LIN {X 0,Y 401.58,Z 643.451,A -85,B 0,C 180,E1 -18913.491,E2 -18913.491} C_VEL
LIN {X 0,Y 402.309,Z 631.628,A -85,B 0,C 180,E1 -18914.623,E2 -18914.623} C_VEL
LIN {X 0,Y 403.111,Z 618.78,A -85,B 0,C 180,E1 -18915.625,E2 -18915.625} C_VEL
LIN {X 0,Y 403.802,Z 604.625,A -85,B 0,C 180,E1 -18916.502,E2 -18916.502} C_VEL
LIN {X 0,Y 404.446,Z 589.348,A -85,B 0,C 180,E1 -18917.22,E2 -18917.22} C_VEL
LIN {X 0,Y 404.999,Z 573.982,A -85,B 0,C 180,E1 -18917.715,E2 -18917.715} C_VEL
LIN {X 0,Y 407.837,Z 472.83,A -85,B 0,C 180,E1 -18920.256,E2 -18920.256} C_VEL
LIN {X 0,Y 405.076,Z 441.864,A -85,B 0,C 180,E1 -18921.136,E2 -18921.136} C_VEL
LIN {X 0,Y 404.994,Z 439.403,A -85,B 0,C 180,E1 -18921.232,E2 -18921.232} C_VEL
LIN {X 0,Y 406.943,Z 410.051,A -85,B 0,C 180,E1 -18925.079,E2 -18925.079} C_VEL
LIN {X 0,Y 408.958,Z 382.784,A -85,B 0,C 180,E1 -18928.658,E2 -18928.658} C_VEL
LIN {X 0,Y 405.49,Z 366.591,A -85,B 0,C 180,E1 -18930.997,E2 -18930.997} C_VEL
LIN {X 0,Y 401.287,Z 348.058,A -85,B 0,C 180,E1 -18933.747,E2 -18933.747} C_VEL
LIN {X 0,Y 401.239,Z 348.061,A -85,B 0,C 180,E1 -18936.58,E2 -18936.58} C_VEL
LIN {X 0,Y 401.222,Z 348.061,A -85,B 0,C 180,E1 -18939.813,E2 -18939.813} C_VEL
LIN {X 0,Y 401.236,Z 348.064,A -85,B 0,C 180,E1 -18942.909,E2 -18942.909} C_VEL
LIN {X 0,Y 401.28,Z 348.053,A -85,B 0,C 180,E1 -18945.716,E2 -18945.716} C_VEL
LIN {X 0,Y 401.214,Z 348.067,A -85,B 0,C 180,E1 -18948.652,E2 -18948.652} C_VEL
LIN {X 0,Y 401.253,Z 348.057,A -85,B 0,C 180,E1 -18951.771,E2 -18951.771} C_VEL
LIN {X 0,Y 401.255,Z 348.059,A -85,B 0,C 180,E1 -18955.13,E2 -18955.13} C_VEL
LIN {X 0,Y 401.243,Z 348.059,A -85,B 0,C 180,E1 -18958.803,E2 -18958.803} C_VEL
LIN {X 0,Y 401.259,Z 348.058,A -85,B 0,C 180,E1 -18961.88,E2 -18961.88} C_VEL
LIN {X 0,Y 401.254,Z 348.058,A -85,B 0,C 180,E1 -18965.232,E2 -18965.232} C_VEL
LIN {X 0,Y 401.256,Z 348.062,A -85,B 0,C 180,E1 -18968.495,E2 -18968.495} C_VEL
LIN {X 0,Y 401.293,Z 348.058,A -85,B 0,C 180,E1 -18971.689,E2 -18971.689} C_VEL
LIN {X 0,Y 401.284,Z 348.059,A -85,B 0,C 180,E1 -18972.24,E2 -18972.24} C_VEL
LIN {X 0,Y 404.072,Z 355.193,A -85,B 0,C 180,E1 -18972.535,E2 -18972.535} C_VEL
LIN {X 0,Y 412.124,Z 375.34,A -85,B 0,C 180,E1 -18973.336,E2 -18973.336} C_VEL
LIN {X 0,Y 410.823,Z 454.396,A -85,B 0,C 180,E1 -18974.708,E2 -18974.708} C_VEL
LIN {X 0,Y 410.699,Z 471.641,A -85,B 0,C 180,E1 -18975.083,E2 -18975.083} C_VEL
LIN {X 0,Y 410.292,Z 486.19,A -85,B 0,C 180,E1 -18975.605,E2 -18975.605} C_VEL
LIN {X 0,Y 409.658,Z 499.427,A -85,B 0,C 180,E1 -18976.276,E2 -18976.276} C_VEL
LIN {X 0,Y 408.783,Z 512.277,A -85,B 0,C 180,E1 -18977.129,E2 -18977.129} C_VEL
LIN {X 0,Y 407.855,Z 525.041,A -85,B 0,C 180,E1 -18978.214,E2 -18978.214} C_VEL
LIN {X 0,Y 406.772,Z 536.867,A -85,B 0,C 180,E1 -18979.458,E2 -18979.458} C_VEL
LIN {X 0,Y 405.528,Z 547.412,A -85,B 0,C 180,E1 -18980.807,E2 -18980.807} C_VEL
LIN {X 0,Y 404.408,Z 556.91,A -85,B 0,C 180,E1 -18982.286,E2 -18982.286} C_VEL
LIN {X 0,Y 403.349,Z 564.807,A -85,B 0,C 180,E1 -18983.769,E2 -18983.769} C_VEL
LIN {X 0,Y 402.397,Z 572.372,A -85,B 0,C 180,E1 -18985.508,E2 -18985.508} C_VEL
LIN {X 0,Y 401.791,Z 577.649,A -85,B 0,C 180,E1 -18987.002,E2 -18987.002} C_VEL
LIN {X 0,Y 401.183,Z 583.211,A -85,B 0,C 180,E1 -18989,E2 -18989} C_VEL
LIN {X 0,Y 400.805,Z 587.257,A -85,B 0,C 180,E1 -18991.002,E2 -18991.002} C_VEL
LIN {X 0,Y 400.584,Z 589.922,A -85,B 0,C 180,E1 -18993.007,E2 -18993.007} C_VEL
LIN {X 0,Y 400.657,Z 591.257,A -85,B 0,C 180,E1 -18995.015,E2 -18995.015} C_VEL
LIN {X 0,Y 400.827,Z 591.305,A -85,B 0,C 180,E1 -18997.026,E2 -18997.026} C_VEL
LIN {X 0,Y 401.166,Z 590.052,A -85,B 0,C 180,E1 -18999.041,E2 -18999.041} C_VEL
LIN {X 0,Y 401.726,Z 587.461,A -85,B 0,C 180,E1 -19001.058,E2 -19001.058} C_VEL
LIN {X 0,Y 402.683,Z 583.437,A -85,B 0,C 180,E1 -19003.069,E2 -19003.069} C_VEL
LIN {X 0,Y 403.855,Z 577.868,A -85,B 0,C 180,E1 -19005.08,E2 -19005.08} C_VEL
LIN {X 0,Y 404.901,Z 572.55,A -85,B 0,C 180,E1 -19006.585,E2 -19006.585} C_VEL
LIN {X 0,Y 406.377,Z 564.566,A -85,B 0,C 180,E1 -19008.407,E2 -19008.407} C_VEL
LIN {X 0,Y 408.022,Z 555.415,A -85,B 0,C 180,E1 -19010.081,E2 -19010.081} C_VEL
LIN {X 0,Y 409.614,Z 545.412,A -85,B 0,C 180,E1 -19011.571,E2 -19011.571} C_VEL
LIN {X 0,Y 411.2,Z 534.021,A -85,B 0,C 180,E1 -19012.948,E2 -19012.948} C_VEL
LIN {X 0,Y 412.585,Z 522.901,A -85,B 0,C 180,E1 -19014.045,E2 -19014.045} C_VEL
LIN {X 0,Y 413.931,Z 510.55,A -85,B 0,C 180,E1 -19015.027,E2 -19015.027} C_VEL
LIN {X 0,Y 414.787,Z 497.822,A -85,B 0,C 180,E1 -19015.842,E2 -19015.842} C_VEL
LIN {X 0,Y 415.567,Z 483.487,A -85,B 0,C 180,E1 -19016.527,E2 -19016.527} C_VEL
LIN {X 0,Y 415.988,Z 469.059,A -85,B 0,C 180,E1 -19017.004,E2 -19017.004} C_VEL
LIN {X 0,Y 416.665,Z 431.837,A -85,B 0,C 180,E1 -19017.69,E2 -19017.69} C_VEL
LIN {X 0,Y 416.122,Z 426.037,A -85,B 0,C 180,E1 -19017.834,E2 -19017.834} C_VEL
LIN {X 0,Y 411.482,Z 407.365,A -85,B 0,C 180,E1 -19018.5,E2 -19018.5} C_VEL
LIN {X 0,Y 411.102,Z 401.561,A -85,B 0,C 180,E1 -19018.638,E2 -19018.638} C_VEL
LIN {X 0,Y 411.271,Z 385.01,A -85,B 0,C 180,E1 -19018.943,E2 -19018.943} C_VEL
LIN {X 0,Y 402.695,Z 366.36,A -85,B 0,C 180,E1 -19019.927,E2 -19019.927} C_VEL
LIN {X 0,Y 394.318,Z 349.692,A -85,B 0,C 180,E1 -19020.909,E2 -19020.909} C_VEL
LIN {X 0,Y 394.183,Z 348.941,A -85,B 0,C 180,E1 -19020.969,E2 -19020.969} C_VEL
LIN {X 0,Y 394.127,Z 348.949,A -85,B 0,C 180,E1 -19024.66,E2 -19024.66} C_VEL
LIN {X 0,Y 394.153,Z 348.945,A -85,B 0,C 180,E1 -19027.172,E2 -19027.172} C_VEL
LIN {X 0,Y 394.132,Z 348.949,A -85,B 0,C 180,E1 -19030.165,E2 -19030.165} C_VEL
LIN {X 0,Y 394.138,Z 348.951,A -85,B 0,C 180,E1 -19033.876,E2 -19033.876} C_VEL
LIN {X 0,Y 394.145,Z 348.946,A -85,B 0,C 180,E1 -19036.771,E2 -19036.771} C_VEL
LIN {X 0,Y 394.134,Z 348.944,A -85,B 0,C 180,E1 -19040.224,E2 -19040.224} C_VEL
LIN {X 0,Y 394.148,Z 348.906,A -85,B 0,C 180,E1 -19043.102,E2 -19043.102} C_VEL
LIN {X 0,Y 394.15,Z 348.941,A -85,B 0,C 180,E1 -19046.641,E2 -19046.641} C_VEL
LIN {X 0,Y 394.173,Z 348.935,A -85,B 0,C 180,E1 -19050.161,E2 -19050.161} C_VEL
LIN {X 0,Y 394.207,Z 348.929,A -85,B 0,C 180,E1 -19053.627,E2 -19053.627} C_VEL
LIN {X 0,Y 394.168,Z 348.942,A -85,B 0,C 180,E1 -19056.986,E2 -19056.986} C_VEL
LIN {X 0,Y 394.202,Z 348.929,A -85,B 0,C 180,E1 -19058.535,E2 -19058.535} C_VEL
LIN {X 0,Y 400.317,Z 371.331,A -85,B 0,C 180,E1 -19059.301,E2 -19059.301} C_VEL
LIN {X 0,Y 398.077,Z 464.711,A -85,B 0,C 180,E1 -19061.671,E2 -19061.671} C_VEL
LIN {X 0,Y 397.816,Z 479.463,A -85,B 0,C 180,E1 -19062.218,E2 -19062.218} C_VEL
LIN {X 0,Y 397.322,Z 493.984,A -85,B 0,C 180,E1 -19062.957,E2 -19062.957} C_VEL
LIN {X 0,Y 396.777,Z 507.71,A -85,B 0,C 180,E1 -19063.856,E2 -19063.856} C_VEL
LIN {X 0,Y 396.137,Z 520.276,A -85,B 0,C 180,E1 -19064.882,E2 -19064.882} C_VEL
LIN {X 0,Y 395.506,Z 533.102,A -85,B 0,C 180,E1 -19066.167,E2 -19066.167} C_VEL
LIN {X 0,Y 395.015,Z 544.496,A -85,B 0,C 180,E1 -19067.548,E2 -19067.548} C_VEL
LIN {X 0,Y 394.447,Z 554.452,A -85,B 0,C 180,E1 -19068.995,E2 -19068.995} C_VEL
LIN {X 0,Y 393.925,Z 563.283,A -85,B 0,C 180,E1 -19070.533,E2 -19070.533} C_VEL
LIN {X 0,Y 393.535,Z 571.747,A -85,B 0,C 180,E1 -19072.328,E2 -19072.328} C_VEL
LIN {X 0,Y 393.339,Z 577.712,A -85,B 0,C 180,E1 -19073.866,E2 -19073.866} C_VEL
LIN {X 0,Y 393.339,Z 584.025,A -85,B 0,C 180,E1 -19075.915,E2 -19075.915} C_VEL
LIN {X 0,Y 393.351,Z 587.625,A -85,B 0,C 180,E1 -19077.448,E2 -19077.448} C_VEL
LIN {X 0,Y 393.465,Z 590.375,A -85,B 0,C 180,E1 -19078.98,E2 -19078.98} C_VEL
LIN {X 0,Y 393.85,Z 592.716,A -85,B 0,C 180,E1 -19081.019,E2 -19081.019} C_VEL
LIN {X 0,Y 394.504,Z 593.628,A -85,B 0,C 180,E1 -19083.053,E2 -19083.053} C_VEL
LIN {X 0,Y 395.419,Z 593.116,A -85,B 0,C 180,E1 -19085.081,E2 -19085.081} C_VEL
LIN {X 0,Y 396.591,Z 591.142,A -85,B 0,C 180,E1 -19087.101,E2 -19087.101} C_VEL
LIN {X 0,Y 397.274,Z 589.601,A -85,B 0,C 180,E1 -19088.108,E2 -19088.108} C_VEL
LIN {X 0,Y 399.178,Z 585.289,A -85,B 0,C 180,E1 -19090.106,E2 -19090.106} C_VEL
LIN {X 0,Y 400.768,Z 580.992,A -85,B 0,C 180,E1 -19091.595,E2 -19091.595} C_VEL
LIN {X 0,Y 402.678,Z 574.711,A -85,B 0,C 180,E1 -19093.325,E2 -19093.325} C_VEL
LIN {X 0,Y 404.905,Z 566.861,A -85,B 0,C 180,E1 -19095.039,E2 -19095.039} C_VEL
LIN {X 0,Y 406.955,Z 558.64,A -85,B 0,C 180,E1 -19096.499,E2 -19096.499} C_VEL
LIN {X 0,Y 409.19,Z 548.719,A -85,B 0,C 180,E1 -19097.946,E2 -19097.946} C_VEL
LIN {X 0,Y 411.656,Z 536.579,A -85,B 0,C 180,E1 -19099.378,E2 -19099.378} C_VEL
LIN {X 0,Y 413.904,Z 524.167,A -85,B 0,C 180,E1 -19100.557,E2 -19100.557} C_VEL
LIN {X 0,Y 415.905,Z 509.912,A -85,B 0,C 180,E1 -19101.651,E2 -19101.651} C_VEL
LIN {X 0,Y 417.437,Z 495.791,A -85,B 0,C 180,E1 -19102.508,E2 -19102.508} C_VEL
LIN {X 0,Y 418.537,Z 482.493,A -85,B 0,C 180,E1 -19103.123,E2 -19103.123} C_VEL
LIN {X 0,Y 419.857,Z 461.411,A -85,B 0,C 180,E1 -19103.831,E2 -19103.831} C_VEL
LIN {X 0,Y 425.647,Z 397.413,A -85,B 0,C 180,E1 -19105.699,E2 -19105.699} C_VEL
LIN {X 0,Y 420.947,Z 388.333,A -85,B 0,C 180,E1 -19106.87,E2 -19106.87} C_VEL
LIN {X 0,Y 415.066,Z 378.237,A -85,B 0,C 180,E1 -19108.46,E2 -19108.46} C_VEL
LIN {X 0,Y 411.495,Z 373.014,A -85,B 0,C 180,E1 -19109.492,E2 -19109.492} C_VEL
LIN {X 0,Y 408.951,Z 369.218,A -85,B 0,C 180,E1 -19110.302,E2 -19110.302} C_VEL
LIN {X 0,Y 406.363,Z 365.403,A -85,B 0,C 180,E1 -19111.188,E2 -19111.188} C_VEL
LIN {X 0,Y 403.453,Z 361.802,A -85,B 0,C 180,E1 -19112.251,E2 -19112.251} C_VEL
LIN {X 0,Y 402.379,Z 359.935,A -85,B 0,C 180,E1 -19112.701,E2 -19112.701} C_VEL
LIN {X 0,Y 399.857,Z 357.401,A -85,B 0,C 180,E1 -19113.756,E2 -19113.756} C_VEL
LIN {X 0,Y 398.478,Z 354.589,A -85,B 0,C 180,E1 -19114.493,E2 -19114.493} C_VEL
LIN {X 0,Y 395.991,Z 352.852,A -85,B 0,C 180,E1 -19115.712,E2 -19115.712} C_VEL
LIN {X 0,Y 394.311,Z 349.707,A -85,B 0,C 180,E1 -19117.154,E2 -19117.154} C_VEL
LIN {X 0,Y 394.188,Z 348.932,A -85,B 0,C 180,E1 -19117.488,E2 -19117.488} C_VEL
LIN {X 0,Y 394.141,Z 348.938,A -85,B 0,C 180,E1 -19121.113,E2 -19121.113} C_VEL
LIN {X 0,Y 394.174,Z 348.938,A -85,B 0,C 180,E1 -19124.7,E2 -19124.7} C_VEL
LIN {X 0,Y 394.149,Z 348.943,A -85,B 0,C 180,E1 -19128.278,E2 -19128.278} C_VEL
LIN {X 0,Y 394.165,Z 349.108,A -85,B 0,C 180,E1 -19129.409,E2 -19129.409} C_VEL
LIN {X 0,Y 395.196,Z 351.875,A -85,B 0,C 180,E1 -19130.436,E2 -19130.436} C_VEL
LIN {X 0,Y 397.598,Z 354.181,A -85,B 0,C 180,E1 -19131.854,E2 -19131.854} C_VEL
LIN {X 0,Y 398.536,Z 354.801,A -85,B 0,C 180,E1 -19132.321,E2 -19132.321} C_VEL
LIN {X 0,Y 399.934,Z 357.773,A -85,B 0,C 180,E1 -19133.146,E2 -19133.146} C_VEL
LIN {X 0,Y 400.838,Z 359.111,A -85,B 0,C 180,E1 -19133.603,E2 -19133.603} C_VEL
LIN {X 0,Y 405.1,Z 371.833,A -85,B 0,C 180,E1 -19135.918,E2 -19135.918} C_VEL
LIN {X 0,Y 409.584,Z 385.954,A -85,B 0,C 180,E1 -19137.895,E2 -19137.895} C_VEL
LIN {X 0,Y 410.898,Z 390.124,A -85,B 0,C 180,E1 -19138.422,E2 -19138.422} C_VEL
LIN {X 0,Y 412.58,Z 396.205,A -85,B 0,C 180,E1 -19139.099,E2 -19139.099} C_VEL
LIN {X 0,Y 414.9,Z 416.547,A -85,B 0,C 180,E1 -19140.564,E2 -19140.564} C_VEL
LIN {X 0,Y 417.082,Z 438.07,A -85,B 0,C 180,E1 -19141.924,E2 -19141.924} C_VEL
LIN {X 0,Y 418.558,Z 458.629,A -85,B 0,C 180,E1 -19143.047,E2 -19143.047} C_VEL
LIN {X 0,Y 419,Z 480.558,A -85,B 0,C 180,E1 -19144.021,E2 -19144.021} C_VEL
LIN {X 0,Y 416.342,Z 513.747,A -85,B 0,C 180,E1 -19144.995,E2 -19144.995} C_VEL
LIN {X 0,Y 413.523,Z 547.21,A -85,B 0,C 180,E1 -19145.98,E2 -19145.98} C_VEL
LIN {X 0,Y 411.488,Z 563.008,A -85,B 0,C 180,E1 -19146.62,E2 -19146.62} C_VEL
LIN {X 0,Y 408.946,Z 578.628,A -85,B 0,C 180,E1 -19147.465,E2 -19147.465} C_VEL
LIN {X 0,Y 406.192,Z 593.435,A -85,B 0,C 180,E1 -19148.504,E2 -19148.504} C_VEL
LIN {X 0,Y 403.496,Z 606.656,A -85,B 0,C 180,E1 -19149.684,E2 -19149.684} C_VEL
LIN {X 0,Y 400.718,Z 619.767,A -85,B 0,C 180,E1 -19151.133,E2 -19151.133} C_VEL
LIN {X 0,Y 398.386,Z 630.692,A -85,B 0,C 180,E1 -19152.609,E2 -19152.609} C_VEL
LIN {X 0,Y 396.45,Z 639.832,A -85,B 0,C 180,E1 -19154.106,E2 -19154.106} C_VEL
LIN {X 0,Y 394.809,Z 648.723,A -85,B 0,C 180,E1 -19155.88,E2 -19155.88} C_VEL
LIN {X 0,Y 393.743,Z 656.054,A -85,B 0,C 180,E1 -19157.674,E2 -19157.674} C_VEL
LIN {X 0,Y 393.485,Z 658.116,A -85,B 0,C 180,E1 -19158.171,E2 -19158.171} C_VEL
LIN {X 0,Y 392.987,Z 667.205,A -85,B 0,C 180,E1 -19159.473,E2 -19159.473} C_VEL
LIN {X 0,Y 392.568,Z 676.261,A -85,B 0,C 180,E1 -19161.018,E2 -19161.018} C_VEL
LIN {X 0,Y 392.231,Z 684.852,A -85,B 0,C 180,E1 -19162.819,E2 -19162.819} C_VEL
LIN {X 0,Y 392.082,Z 690.842,A -85,B 0,C 180,E1 -19164.361,E2 -19164.361} C_VEL
LIN {X 0,Y 391.975,Z 695.673,A -85,B 0,C 180,E1 -19165.901,E2 -19165.901} C_VEL
LIN {X 0,Y 391.913,Z 699.461,A -85,B 0,C 180,E1 -19167.439,E2 -19167.439} C_VEL
LIN {X 0,Y 391.91,Z 702.341,A -85,B 0,C 180,E1 -19168.976,E2 -19168.976} C_VEL
LIN {X 0,Y 391.919,Z 703.757,A -85,B 0,C 180,E1 -19170,E2 -19170} C_VEL
LIN {X 0,Y 391.891,Z 705.465,A -85,B 0,C 180,E1 -19172.048,E2 -19172.048} C_VEL
LIN {X 0,Y 391.96,Z 705.706,A -85,B 0,C 180,E1 -19174.099,E2 -19174.099} C_VEL
LIN {X 0,Y 392.331,Z 704.501,A -85,B 0,C 180,E1 -19176.149,E2 -19176.149} C_VEL
LIN {X 0,Y 393.018,Z 701.849,A -85,B 0,C 180,E1 -19178.197,E2 -19178.197} C_VEL
LIN {X 0,Y 393.984,Z 697.662,A -85,B 0,C 180,E1 -19180.241,E2 -19180.241} C_VEL
LIN {X 0,Y 395.723,Z 691.846,A -85,B 0,C 180,E1 -19182.263,E2 -19182.263} C_VEL
LIN {X 0,Y 397.333,Z 684.798,A -85,B 0,C 180,E1 -19184.17,E2 -19184.17} C_VEL
LIN {X 0,Y 399.284,Z 677.293,A -85,B 0,C 180,E1 -19185.778,E2 -19185.778} C_VEL
LIN {X 0,Y 401.742,Z 667.387,A -85,B 0,C 180,E1 -19187.503,E2 -19187.503} C_VEL
LIN {X 0,Y 404.089,Z 657.084,A -85,B 0,C 180,E1 -19188.966,E2 -19188.966} C_VEL
LIN {X 0,Y 406.809,Z 644.673,A -85,B 0,C 180,E1 -19190.406,E2 -19190.406} C_VEL
LIN {X 0,Y 409.335,Z 632.032,A -85,B 0,C 180,E1 -19191.586,E2 -19191.586} C_VEL
LIN {X 0,Y 411.507,Z 619.821,A -85,B 0,C 180,E1 -19192.518,E2 -19192.518} C_VEL
LIN {X 0,Y 413.893,Z 604.525,A -85,B 0,C 180,E1 -19193.434,E2 -19193.434} C_VEL
LIN {X 0,Y 415.936,Z 589.429,A -85,B 0,C 180,E1 -19194.103,E2 -19194.103} C_VEL
LIN {X 0,Y 418.104,Z 566.637,A -85,B 0,C 180,E1 -19194.816,E2 -19194.816} C_VEL
LIN {X 0,Y 425.848,Z 486.064,A -85,B 0,C 180,E1 -19197.224,E2 -19197.224} C_VEL
LIN {X 0,Y 426.185,Z 476.939,A -85,B 0,C 180,E1 -19197.591,E2 -19197.591} C_VEL
LIN {X 0,Y 425.687,Z 457.567,A -85,B 0,C 180,E1 -19198.602,E2 -19198.602} C_VEL
LIN {X 0,Y 424.826,Z 444.628,A -85,B 0,C 180,E1 -19199.408,E2 -19199.408} C_VEL
LIN {X 0,Y 424.35,Z 436.844,A -85,B 0,C 180,E1 -19199.955,E2 -19199.955} C_VEL
LIN {X 0,Y 426.009,Z 420.687,A -85,B 0,C 180,E1 -19201.593,E2 -19201.593} C_VEL
LIN {X 0,Y 427.546,Z 409.077,A -85,B 0,C 180,E1 -19202.914,E2 -19202.914} C_VEL
LIN {X 0,Y 427.531,Z 403.537,A -85,B 0,C 180,E1 -19203.851,E2 -19203.851} C_VEL
LIN {X 0,Y 426.297,Z 400.847,A -85,B 0,C 180,E1 -19204.76,E2 -19204.76} C_VEL
LIN {X 0,Y 424.019,Z 397.104,A -85,B 0,C 180,E1 -19206.491,E2 -19206.491} C_VEL
LIN {X 0,Y 422.633,Z 394.946,A -85,B 0,C 180,E1 -19207.822,E2 -19207.822} C_VEL
LIN {X 0,Y 420.894,Z 392.809,A -85,B 0,C 180,E1 -19210.046,E2 -19210.046} C_VEL
LIN {X 0,Y 420.043,Z 392.103,A -85,B 0,C 180,E1 -19211.838,E2 -19211.838} C_VEL
LIN {X 0,Y 419.719,Z 392.284,A -85,B 0,C 180,E1 -19214.143,E2 -19214.143} C_VEL
LIN {X 0,Y 419.855,Z 393.5,A -85,B 0,C 180,E1 -19215.838,E2 -19215.838} C_VEL
LIN {X 0,Y 420.591,Z 396.611,A -85,B 0,C 180,E1 -19218.229,E2 -19218.229} C_VEL
LIN {X 0,Y 421.525,Z 400.483,A -85,B 0,C 180,E1 -19220.238,E2 -19220.238} C_VEL
LIN {X 0,Y 422.633,Z 405.321,A -85,B 0,C 180,E1 -19222.178,E2 -19222.178} C_VEL
LIN {X 0,Y 423.731,Z 411.286,A -85,B 0,C 180,E1 -19224.095,E2 -19224.095} C_VEL
LIN {X 0,Y 424.745,Z 419.525,A -85,B 0,C 180,E1 -19226.25,E2 -19226.25} C_VEL
LIN {X 0,Y 424.873,Z 421.549,A -85,B 0,C 180,E1 -19226.716,E2 -19226.716} C_VEL
LIN {X 0,Y 420.776,Z 439.481,A -85,B 0,C 180,E1 -19229.434,E2 -19229.434} C_VEL
LIN {X 0,Y 423.204,Z 456.319,A -85,B 0,C 180,E1 -19230.818,E2 -19230.818} C_VEL
LIN {X 0,Y 425.126,Z 471.437,A -85,B 0,C 180,E1 -19231.888,E2 -19231.888} C_VEL
LIN {X 0,Y 426.272,Z 485.082,A -85,B 0,C 180,E1 -19232.701,E2 -19232.701} C_VEL
LIN {X 0,Y 418.787,Z 563.538,A -85,B 0,C 180,E1 -19235.019,E2 -19235.019} C_VEL
LIN {X 0,Y 416.753,Z 585.213,A -85,B 0,C 180,E1 -19235.684,E2 -19235.684} C_VEL
LIN {X 0,Y 414.717,Z 600.648,A -85,B 0,C 180,E1 -19236.351,E2 -19236.351} C_VEL
LIN {X 0,Y 412.612,Z 614.555,A -85,B 0,C 180,E1 -19237.15,E2 -19237.15} C_VEL
LIN {X 0,Y 410.394,Z 627.255,A -85,B 0,C 180,E1 -19238.078,E2 -19238.078} C_VEL
LIN {X 0,Y 407.829,Z 640.307,A -85,B 0,C 180,E1 -19239.254,E2 -19239.254} C_VEL
LIN {X 0,Y 405.259,Z 652.194,A -85,B 0,C 180,E1 -19240.567,E2 -19240.567} C_VEL
LIN {X 0,Y 402.728,Z 663,A -85,B 0,C 180,E1 -19242.018,E2 -19242.018} C_VEL
LIN {X 0,Y 400.549,Z 671.981,A -85,B 0,C 180,E1 -19243.491,E2 -19243.491} C_VEL
LIN {X 0,Y 398.442,Z 680.08,A -85,B 0,C 180,E1 -19245.089,E2 -19245.089} C_VEL
LIN {X 0,Y 396.813,Z 686.833,A -85,B 0,C 180,E1 -19246.734,E2 -19246.734} C_VEL
LIN {X 0,Y 395.371,Z 691.981,A -85,B 0,C 180,E1 -19248.245,E2 -19248.245} C_VEL
LIN {X 0,Y 393.93,Z 697.271,A -85,B 0,C 180,E1 -19250.275,E2 -19250.275} C_VEL
LIN {X 0,Y 393.122,Z 700.254,A -85,B 0,C 180,E1 -19251.805,E2 -19251.805} C_VEL
LIN {X 0,Y 392.364,Z 702.892,A -85,B 0,C 180,E1 -19253.851,E2 -19253.851} C_VEL
LIN {X 0,Y 391.948,Z 704.083,A -85,B 0,C 180,E1 -19255.901,E2 -19255.901} C_VEL
LIN {X 0,Y 391.803,Z 703.841,A -85,B 0,C 180,E1 -19257.951,E2 -19257.951} C_VEL
LIN {X 0,Y 391.821,Z 702.153,A -85,B 0,C 180,E1 -19260,E2 -19260} C_VEL
LIN {X 0,Y 391.848,Z 698.975,A -85,B 0,C 180,E1 -19262.049,E2 -19262.049} C_VEL
LIN {X 0,Y 391.881,Z 695.519,A -85,B 0,C 180,E1 -19263.587,E2 -19263.587} C_VEL
LIN {X 0,Y 391.993,Z 691.113,A -85,B 0,C 180,E1 -19265.126,E2 -19265.126} C_VEL
LIN {X 0,Y 392.192,Z 684.591,A -85,B 0,C 180,E1 -19266.924,E2 -19266.924} C_VEL
LIN {X 0,Y 392.518,Z 676.425,A -85,B 0,C 180,E1 -19268.725,E2 -19268.725} C_VEL
LIN {X 0,Y 392.94,Z 667.866,A -85,B 0,C 180,E1 -19270.269,E2 -19270.269} C_VEL
LIN {X 0,Y 393.625,Z 657.306,A -85,B 0,C 180,E1 -19271.844,E2 -19271.844} C_VEL
LIN {X 0,Y 394.334,Z 646.08,A -85,B 0,C 180,E1 -19273.221,E2 -19273.221} C_VEL
LIN {X 0,Y 395.082,Z 633.392,A -85,B 0,C 180,E1 -19274.503,E2 -19274.503} C_VEL
LIN {X 0,Y 395.913,Z 621.035,A -85,B 0,C 180,E1 -19275.521,E2 -19275.521} C_VEL
LIN {X 0,Y 396.666,Z 607.579,A -85,B 0,C 180,E1 -19276.412,E2 -19276.412} C_VEL
LIN {X 0,Y 397.25,Z 593.912,A -85,B 0,C 180,E1 -19277.112,E2 -19277.112} C_VEL
LIN {X 0,Y 397.813,Z 578.573,A -85,B 0,C 180,E1 -19277.683,E2 -19277.683} C_VEL
LIN {X 0,Y 400.841,Z 473.137,A -85,B 0,C 180,E1 -19280.423,E2 -19280.423} C_VEL
LIN {X 0,Y 398.096,Z 441.756,A -85,B 0,C 180,E1 -19281.333,E2 -19281.333} C_VEL
LIN {X 0,Y 398.002,Z 439.421,A -85,B 0,C 180,E1 -19281.426,E2 -19281.426} C_VEL
LIN {X 0,Y 399.917,Z 411.459,A -85,B 0,C 180,E1 -19285.134,E2 -19285.134} C_VEL
LIN {X 0,Y 401.909,Z 385.067,A -85,B 0,C 180,E1 -19288.638,E2 -19288.638} C_VEL
LIN {X 0,Y 401.665,Z 382.149,A -85,B 0,C 180,E1 -19289.048,E2 -19289.048} C_VEL
LIN {X 0,Y 396.805,Z 360.231,A -85,B 0,C 180,E1 -19292.274,E2 -19292.274} C_VEL
LIN {X 0,Y 394.258,Z 348.932,A -85,B 0,C 180,E1 -19293.988,E2 -19293.988} C_VEL
LIN {X 0,Y 394.184,Z 348.945,A -85,B 0,C 180,E1 -19297.169,E2 -19297.169} C_VEL
LIN {X 0,Y 394.169,Z 348.938,A -85,B 0,C 180,E1 -19300.171,E2 -19300.171} C_VEL
LIN {X 0,Y 394.222,Z 348.933,A -85,B 0,C 180,E1 -19303.864,E2 -19303.864} C_VEL
LIN {X 0,Y 394.181,Z 348.941,A -85,B 0,C 180,E1 -19306.766,E2 -19306.766} C_VEL
LIN {X 0,Y 394.175,Z 348.938,A -85,B 0,C 180,E1 -19310.229,E2 -19310.229} C_VEL
LIN {X 0,Y 394.187,Z 348.938,A -85,B 0,C 180,E1 -19313.095,E2 -19313.095} C_VEL
LIN {X 0,Y 394.2,Z 348.936,A -85,B 0,C 180,E1 -19315.347,E2 -19315.347} C_VEL
LIN {X 0,Y 394.192,Z 348.937,A -85,B 0,C 180,E1 -19318.982,E2 -19318.982} C_VEL
LIN {X 0,Y 394.202,Z 348.936,A -85,B 0,C 180,E1 -19321.331,E2 -19321.331} C_VEL
LIN {X 0,Y 394.221,Z 348.937,A -85,B 0,C 180,E1 -19324.759,E2 -19324.759} C_VEL
LIN {X 0,Y 394.236,Z 348.937,A -85,B 0,C 180,E1 -19328.093,E2 -19328.093} C_VEL
LIN {X 0,Y 394.248,Z 348.934,A -85,B 0,C 180,E1 -19331.349,E2 -19331.349} C_VEL
LIN {X 0,Y 394.274,Z 348.932,A -85,B 0,C 180,E1 -19331.856,E2 -19331.856} C_VEL
LIN {X 0,Y 396.093,Z 353.868,A -85,B 0,C 180,E1 -19332.061,E2 -19332.061} C_VEL
LIN {X 0,Y 404.56,Z 374.582,A -85,B 0,C 180,E1 -19332.923,E2 -19332.923} C_VEL
LIN {X 0,Y 405.468,Z 377.593,A -85,B 0,C 180,E1 -19333.028,E2 -19333.028} C_VEL
LIN {X 0,Y 404.111,Z 454.603,A -85,B 0,C 180,E1 -19334.383,E2 -19334.383} C_VEL
LIN {X 0,Y 403.987,Z 472.045,A -85,B 0,C 180,E1 -19334.765,E2 -19334.765} C_VEL
LIN {X 0,Y 403.618,Z 485.956,A -85,B 0,C 180,E1 -19335.265,E2 -19335.265} C_VEL
LIN {X 0,Y 402.922,Z 500.013,A -85,B 0,C 180,E1 -19335.978,E2 -19335.978} C_VEL
LIN {X 0,Y 402.071,Z 512.075,A -85,B 0,C 180,E1 -19336.783,E2 -19336.783} C_VEL
LIN {X 0,Y 401.224,Z 523.947,A -85,B 0,C 180,E1 -19337.78,E2 -19337.78} C_VEL
LIN {X 0,Y 400.127,Z 535.967,A -85,B 0,C 180,E1 -19339.026,E2 -19339.026} C_VEL
LIN {X 0,Y 398.828,Z 546.791,A -85,B 0,C 180,E1 -19340.396,E2 -19340.396} C_VEL
LIN {X 0,Y 397.608,Z 556.526,A -85,B 0,C 180,E1 -19341.898,E2 -19341.898} C_VEL
LIN {X 0,Y 396.372,Z 565.823,A -85,B 0,C 180,E1 -19343.659,E2 -19343.659} C_VEL
LIN {X 0,Y 395.39,Z 573.343,A -85,B 0,C 180,E1 -19345.428,E2 -19345.428} C_VEL
LIN {X 0,Y 394.774,Z 578.578,A -85,B 0,C 180,E1 -19346.949,E2 -19346.949} C_VEL
LIN {X 0,Y 394.129,Z 584.106,A -85,B 0,C 180,E1 -19348.982,E2 -19348.982} C_VEL
LIN {X 0,Y 393.768,Z 588.114,A -85,B 0,C 180,E1 -19351.019,E2 -19351.019} C_VEL
LIN {X 0,Y 393.522,Z 590.748,A -85,B 0,C 180,E1 -19353.061,E2 -19353.061} C_VEL
LIN {X 0,Y 393.599,Z 592.044,A -85,B 0,C 180,E1 -19355.105,E2 -19355.105} C_VEL
LIN {X 0,Y 393.787,Z 592.053,A -85,B 0,C 180,E1 -19357.153,E2 -19357.153} C_VEL
LIN {X 0,Y 394.145,Z 590.765,A -85,B 0,C 180,E1 -19359.204,E2 -19359.204} C_VEL
LIN {X 0,Y 394.774,Z 588.138,A -85,B 0,C 180,E1 -19361.255,E2 -19361.255} C_VEL
LIN {X 0,Y 395.763,Z 584.079,A -85,B 0,C 180,E1 -19363.302,E2 -19363.302} C_VEL
LIN {X 0,Y 396.988,Z 578.473,A -85,B 0,C 180,E1 -19365.347,E2 -19365.347} C_VEL
LIN {X 0,Y 398.068,Z 573.114,A -85,B 0,C 180,E1 -19366.878,E2 -19366.878} C_VEL
LIN {X 0,Y 399.561,Z 565.462,A -85,B 0,C 180,E1 -19368.65,E2 -19368.65} C_VEL
LIN {X 0,Y 401.047,Z 557.348,A -85,B 0,C 180,E1 -19370.178,E2 -19370.178} C_VEL
LIN {X 0,Y 402.7,Z 547.584,A -85,B 0,C 180,E1 -19371.692,E2 -19371.692} C_VEL
LIN {X 0,Y 404.338,Z 536.672,A -85,B 0,C 180,E1 -19373.078,E2 -19373.078} C_VEL
LIN {X 0,Y 405.733,Z 526.088,A -85,B 0,C 180,E1 -19374.179,E2 -19374.179} C_VEL
LIN {X 0,Y 407.156,Z 514.033,A -85,B 0,C 180,E1 -19375.2,E2 -19375.2} C_VEL
LIN {X 0,Y 408.114,Z 501.03,A -85,B 0,C 180,E1 -19376.091,E2 -19376.091} C_VEL
LIN {X 0,Y 408.992,Z 486.782,A -85,B 0,C 180,E1 -19376.817,E2 -19376.817} C_VEL
LIN {X 0,Y 409.512,Z 472.533,A -85,B 0,C 180,E1 -19377.328,E2 -19377.328} C_VEL
LIN {X 0,Y 409.774,Z 455.905,A -85,B 0,C 180,E1 -19377.691,E2 -19377.691} C_VEL
LIN {X 0,Y 411.102,Z 401.561,A -85,B 0,C 180,E1 -19378.638,E2 -19378.638} C_VEL
LIN {X 0,Y 410.816,Z 397.713,A -85,B 0,C 180,E1 -19378.731,E2 -19378.731} C_VEL
LIN {X 0,Y 409.15,Z 392.259,A -85,B 0,C 180,E1 -19378.953,E2 -19378.953} C_VEL
LIN {X 0,Y 406.582,Z 387.235,A -85,B 0,C 180,E1 -19379.233,E2 -19379.233} C_VEL
LIN {X 0,Y 400.6,Z 377.321,A -85,B 0,C 180,E1 -19379.868,E2 -19379.868} C_VEL
LIN {X 0,Y 398.946,Z 373.795,A -85,B 0,C 180,E1 -19380.063,E2 -19380.063} C_VEL
LIN {X 0,Y 389.91,Z 355.906,A -85,B 0,C 180,E1 -19381.137,E2 -19381.137} C_VEL
LIN {X 0,Y 387.375,Z 351.002,A -85,B 0,C 180,E1 -19381.447,E2 -19381.447} C_VEL
LIN {X 0,Y 387.127,Z 349.819,A -85,B 0,C 180,E1 -19381.523,E2 -19381.523} C_VEL
LIN {X 0,Y 387.11,Z 349.823,A -85,B 0,C 180,E1 -19385.487,E2 -19385.487} C_VEL
LIN {X 0,Y 387.102,Z 349.825,A -85,B 0,C 180,E1 -19388.915,E2 -19388.915} C_VEL
LIN {X 0,Y 387.068,Z 349.828,A -85,B 0,C 180,E1 -19392.102,E2 -19392.102} C_VEL
LIN {X 0,Y 387.125,Z 349.816,A -85,B 0,C 180,E1 -19395.118,E2 -19395.118} C_VEL
LIN {X 0,Y 387.097,Z 349.82,A -85,B 0,C 180,E1 -19397.97,E2 -19397.97} C_VEL
LIN {X 0,Y 387.1,Z 349.814,A -85,B 0,C 180,E1 -19401.085,E2 -19401.085} C_VEL
LIN {X 0,Y 387.113,Z 349.791,A -85,B 0,C 180,E1 -19404.512,E2 -19404.512} C_VEL
LIN {X 0,Y 387.129,Z 349.811,A -85,B 0,C 180,E1 -19408.351,E2 -19408.351} C_VEL
LIN {X 0,Y 387.155,Z 349.817,A -85,B 0,C 180,E1 -19411.94,E2 -19411.94} C_VEL
LIN {X 0,Y 387.137,Z 349.813,A -85,B 0,C 180,E1 -19415.409,E2 -19415.409} C_VEL
LIN {X 0,Y 387.164,Z 349.806,A -85,B 0,C 180,E1 -19418.383,E2 -19418.383} C_VEL
LIN {X 0,Y 393.222,Z 371.441,A -85,B 0,C 180,E1 -19419.129,E2 -19419.129} C_VEL
LIN {X 0,Y 391.977,Z 415.995,A -85,B 0,C 180,E1 -19420.288,E2 -19420.288} C_VEL
LIN {X 0,Y 390.994,Z 468.125,A -85,B 0,C 180,E1 -19421.669,E2 -19421.669} C_VEL
LIN {X 0,Y 390.694,Z 484.166,A -85,B 0,C 180,E1 -19422.322,E2 -19422.322} C_VEL
LIN {X 0,Y 390.194,Z 498.238,A -85,B 0,C 180,E1 -19423.107,E2 -19423.107} C_VEL
LIN {X 0,Y 389.556,Z 511.968,A -85,B 0,C 180,E1 -19424.085,E2 -19424.085} C_VEL
LIN {X 0,Y 388.875,Z 525.279,A -85,B 0,C 180,E1 -19425.26,E2 -19425.26} C_VEL
LIN {X 0,Y 388.252,Z 537.604,A -85,B 0,C 180,E1 -19426.598,E2 -19426.598} C_VEL
LIN {X 0,Y 387.738,Z 548.39,A -85,B 0,C 180,E1 -19428.009,E2 -19428.009} C_VEL
LIN {X 0,Y 387.118,Z 558.399,A -85,B 0,C 180,E1 -19429.575,E2 -19429.575} C_VEL
LIN {X 0,Y 386.636,Z 568.015,A -85,B 0,C 180,E1 -19431.404,E2 -19431.404} C_VEL
LIN {X 0,Y 386.303,Z 575.748,A -85,B 0,C 180,E1 -19433.231,E2 -19433.231} C_VEL
LIN {X 0,Y 386.203,Z 582.76,A -85,B 0,C 180,E1 -19435.318,E2 -19435.318} C_VEL
LIN {X 0,Y 386.276,Z 586.83,A -85,B 0,C 180,E1 -19436.881,E2 -19436.881} C_VEL
LIN {X 0,Y 386.386,Z 590.907,A -85,B 0,C 180,E1 -19438.961,E2 -19438.961} C_VEL
LIN {X 0,Y 386.812,Z 593.442,A -85,B 0,C 180,E1 -19441.037,E2 -19441.037} C_VEL
LIN {X 0,Y 387.485,Z 594.536,A -85,B 0,C 180,E1 -19443.108,E2 -19443.108} C_VEL
LIN {X 0,Y 388.442,Z 594.207,A -85,B 0,C 180,E1 -19445.173,E2 -19445.173} C_VEL
LIN {X 0,Y 389.67,Z 592.458,A -85,B 0,C 180,E1 -19447.228,E2 -19447.228} C_VEL
LIN {X 0,Y 390.392,Z 591.042,A -85,B 0,C 180,E1 -19448.252,E2 -19448.252} C_VEL
LIN {X 0,Y 391.871,Z 588.115,A -85,B 0,C 180,E1 -19449.776,E2 -19449.776} C_VEL
LIN {X 0,Y 393.444,Z 584.305,A -85,B 0,C 180,E1 -19451.293,E2 -19451.293} C_VEL
LIN {X 0,Y 395.74,Z 577.773,A -85,B 0,C 180,E1 -19453.302,E2 -19453.302} C_VEL
LIN {X 0,Y 398.032,Z 570.392,A -85,B 0,C 180,E1 -19455.044,E2 -19455.044} C_VEL
LIN {X 0,Y 400.539,Z 561.27,A -85,B 0,C 180,E1 -19456.771,E2 -19456.771} C_VEL
LIN {X 0,Y 402.898,Z 551.729,A -85,B 0,C 180,E1 -19458.236,E2 -19458.236} C_VEL
LIN {X 0,Y 405.242,Z 541.213,A -85,B 0,C 180,E1 -19459.566,E2 -19459.566} C_VEL
LIN {X 0,Y 407.739,Z 528.311,A -85,B 0,C 180,E1 -19460.883,E2 -19460.883} C_VEL
LIN {X 0,Y 409.871,Z 515.394,A -85,B 0,C 180,E1 -19461.952,E2 -19461.952} C_VEL
LIN {X 0,Y 411.693,Z 500.553,A -85,B 0,C 180,E1 -19462.93,E2 -19462.93} C_VEL
LIN {X 0,Y 413.07,Z 486.473,A -85,B 0,C 180,E1 -19463.644,E2 -19463.644} C_VEL
LIN {X 0,Y 414.317,Z 467.447,A -85,B 0,C 180,E1 -19464.336,E2 -19464.336} C_VEL
LIN {X 0,Y 420.665,Z 400.403,A -85,B 0,C 180,E1 -19466.344,E2 -19466.344} C_VEL
LIN {X 0,Y 415.988,Z 391.45,A -85,B 0,C 180,E1 -19467.586,E2 -19467.586} C_VEL
LIN {X 0,Y 411.299,Z 383.391,A -85,B 0,C 180,E1 -19468.942,E2 -19468.942} C_VEL
LIN {X 0,Y 407.785,Z 378.027,A -85,B 0,C 180,E1 -19470.022,E2 -19470.022} C_VEL
LIN {X 0,Y 405.871,Z 375.124,A -85,B 0,C 180,E1 -19470.667,E2 -19470.667} C_VEL
LIN {X 0,Y 402.983,Z 370.878,A -85,B 0,C 180,E1 -19471.715,E2 -19471.715} C_VEL
LIN {X 0,Y 400.547,Z 367.618,A -85,B 0,C 180,E1 -19472.653,E2 -19472.653} C_VEL
LIN {X 0,Y 399.702,Z 366.245,A -85,B 0,C 180,E1 -19473.039,E2 -19473.039} C_VEL
LIN {X 0,Y 397.176,Z 363.396,A -85,B 0,C 180,E1 -19474.154,E2 -19474.154} C_VEL
LIN {X 0,Y 395.997,Z 361.11,A -85,B 0,C 180,E1 -19474.802,E2 -19474.802} C_VEL
LIN {X 0,Y 393.426,Z 358.928,A -85,B 0,C 180,E1 -19476.172,E2 -19476.172} C_VEL
LIN {X 0,Y 391.792,Z 356.052,A -85,B 0,C 180,E1 -19477.434,E2 -19477.434} C_VEL
LIN {X 0,Y 391.082,Z 355.308,A -85,B 0,C 180,E1 -19477.995,E2 -19477.995} C_VEL
LIN {X 0,Y 388.747,Z 353.564,A -85,B 0,C 180,E1 -19480.82,E2 -19480.82} C_VEL
LIN {X 0,Y 388.274,Z 352.945,A -85,B 0,C 180,E1 -19482.299,E2 -19482.299} C_VEL
LIN {X 0,Y 388.367,Z 352.984,A -85,B 0,C 180,E1 -19484.699,E2 -19484.699} C_VEL
LIN {X 0,Y 390.189,Z 354.83,A -85,B 0,C 180,E1 -19487.774,E2 -19487.774} C_VEL
LIN {X 0,Y 391.909,Z 355.953,A -85,B 0,C 180,E1 -19489.246,E2 -19489.246} C_VEL
LIN {X 0,Y 393.135,Z 358.796,A -85,B 0,C 180,E1 -19490.406,E2 -19490.406} C_VEL
LIN {X 0,Y 396.064,Z 361.473,A -85,B 0,C 180,E1 -19492.085,E2 -19492.085} C_VEL
LIN {X 0,Y 397.724,Z 364.529,A -85,B 0,C 180,E1 -19493.05,E2 -19493.05} C_VEL
LIN {X 0,Y 398.434,Z 366.493,A -85,B 0,C 180,E1 -19493.499,E2 -19493.499} C_VEL
LIN {X 0,Y 401.97,Z 377.738,A -85,B 0,C 180,E1 -19495.516,E2 -19495.516} C_VEL
LIN {X 0,Y 406.212,Z 391.643,A -85,B 0,C 180,E1 -19497.499,E2 -19497.499} C_VEL
LIN {X 0,Y 408.45,Z 400.088,A -85,B 0,C 180,E1 -19498.488,E2 -19498.488} C_VEL
LIN {X 0,Y 410.511,Z 420.73,A -85,B 0,C 180,E1 -19500.003,E2 -19500.003} C_VEL
LIN {X 0,Y 412.376,Z 441.76,A -85,B 0,C 180,E1 -19501.361,E2 -19501.361} C_VEL
LIN {X 0,Y 413.678,Z 463.926,A -85,B 0,C 180,E1 -19502.58,E2 -19502.58} C_VEL
LIN {X 0,Y 413.758,Z 482.975,A -85,B 0,C 180,E1 -19503.42,E2 -19503.42} C_VEL
LIN {X 0,Y 408.074,Z 546.748,A -85,B 0,C 180,E1 -19505.335,E2 -19505.335} C_VEL
LIN {X 0,Y 406.069,Z 561.738,A -85,B 0,C 180,E1 -19505.951,E2 -19505.951} C_VEL
LIN {X 0,Y 403.587,Z 576.321,A -85,B 0,C 180,E1 -19506.744,E2 -19506.744} C_VEL
LIN {X 0,Y 400.612,Z 591.186,A -85,B 0,C 180,E1 -19507.784,E2 -19507.784} C_VEL
LIN {X 0,Y 397.991,Z 603.459,A -85,B 0,C 180,E1 -19508.852,E2 -19508.852} C_VEL
LIN {X 0,Y 395.235,Z 615.707,A -85,B 0,C 180,E1 -19510.165,E2 -19510.165} C_VEL
LIN {X 0,Y 392.874,Z 626.271,A -85,B 0,C 180,E1 -19511.551,E2 -19511.551} C_VEL
LIN {X 0,Y 390.225,Z 637.41,A -85,B 0,C 180,E1 -19513.31,E2 -19513.31} C_VEL
LIN {X 0,Y 388.363,Z 646.577,A -85,B 0,C 180,E1 -19515.107,E2 -19515.107} C_VEL
LIN {X 0,Y 387.04,Z 654.074,A -85,B 0,C 180,E1 -19516.925,E2 -19516.925} C_VEL
LIN {X 0,Y 386.319,Z 659.05,A -85,B 0,C 180,E1 -19518.317,E2 -19518.317} C_VEL
LIN {X 0,Y 385.741,Z 668.98,A -85,B 0,C 180,E1 -19519.802,E2 -19519.802} C_VEL
LIN {X 0,Y 385.343,Z 677.698,A -85,B 0,C 180,E1 -19521.375,E2 -19521.375} C_VEL
LIN {X 0,Y 385.102,Z 685.99,A -85,B 0,C 180,E1 -19523.21,E2 -19523.21} C_VEL
LIN {X 0,Y 384.98,Z 691.746,A -85,B 0,C 180,E1 -19524.78,E2 -19524.78} C_VEL
LIN {X 0,Y 384.879,Z 696.407,A -85,B 0,C 180,E1 -19526.348,E2 -19526.348} C_VEL
LIN {X 0,Y 384.848,Z 700.055,A -85,B 0,C 180,E1 -19527.914,E2 -19527.914} C_VEL
LIN {X 0,Y 384.834,Z 701.965,A -85,B 0,C 180,E1 -19528.957,E2 -19528.957} C_VEL
LIN {X 0,Y 384.836,Z 703.462,A -85,B 0,C 180,E1 -19530,E2 -19530} C_VEL
LIN {X 0,Y 384.797,Z 705.325,A -85,B 0,C 180,E1 -19532.086,E2 -19532.086} C_VEL
LIN {X 0,Y 384.889,Z 705.729,A -85,B 0,C 180,E1 -19534.174,E2 -19534.174} C_VEL
LIN {X 0,Y 385.272,Z 704.692,A -85,B 0,C 180,E1 -19536.262,E2 -19536.262} C_VEL
LIN {X 0,Y 385.984,Z 702.22,A -85,B 0,C 180,E1 -19538.347,E2 -19538.347} C_VEL
LIN {X 0,Y 387.028,Z 698.278,A -85,B 0,C 180,E1 -19540.427,E2 -19540.427} C_VEL
LIN {X 0,Y 388.852,Z 692.676,A -85,B 0,C 180,E1 -19542.483,E2 -19542.483} C_VEL
LIN {X 0,Y 390.505,Z 685.942,A -85,B 0,C 180,E1 -19544.398,E2 -19544.398} C_VEL
LIN {X 0,Y 392.572,Z 678.603,A -85,B 0,C 180,E1 -19546.055,E2 -19546.055} C_VEL
LIN {X 0,Y 395.163,Z 669.022,A -85,B 0,C 180,E1 -19547.804,E2 -19547.804} C_VEL
LIN {X 0,Y 397.599,Z 659.151,A -85,B 0,C 180,E1 -19549.288,E2 -19549.288} C_VEL
LIN {X 0,Y 400.408,Z 647.17,A -85,B 0,C 180,E1 -19550.747,E2 -19550.747} C_VEL
LIN {X 0,Y 403.051,Z 635.124,A -85,B 0,C 180,E1 -19551.94,E2 -19551.94} C_VEL
LIN {X 0,Y 405.565,Z 622.058,A -85,B 0,C 180,E1 -19553.001,E2 -19553.001} C_VEL
LIN {X 0,Y 408.047,Z 607.517,A -85,B 0,C 180,E1 -19553.925,E2 -19553.925} C_VEL
LIN {X 0,Y 410.412,Z 591.497,A -85,B 0,C 180,E1 -19554.683,E2 -19554.683} C_VEL
LIN {X 0,Y 412.288,Z 574.185,A -85,B 0,C 180,E1 -19555.268,E2 -19555.268} C_VEL
LIN {X 0,Y 420.59,Z 491.85,A -85,B 0,C 180,E1 -19557.774,E2 -19557.774} C_VEL
LIN {X 0,Y 421.404,Z 482.715,A -85,B 0,C 180,E1 -19558.086,E2 -19558.086} C_VEL
LIN {X 0,Y 421.391,Z 468.767,A -85,B 0,C 180,E1 -19558.782,E2 -19558.782} C_VEL
LIN {X 0,Y 420.9,Z 453.135,A -85,B 0,C 180,E1 -19559.687,E2 -19559.687} C_VEL
LIN {X 0,Y 419.933,Z 437.095,A -85,B 0,C 180,E1 -19560.815,E2 -19560.815} C_VEL
LIN {X 0,Y 421.712,Z 422.758,A -85,B 0,C 180,E1 -19562.328,E2 -19562.328} C_VEL
LIN {X 0,Y 423.232,Z 412.625,A -85,B 0,C 180,E1 -19563.509,E2 -19563.509} C_VEL
LIN {X 0,Y 423.265,Z 408.566,A -85,B 0,C 180,E1 -19564.239,E2 -19564.239} C_VEL
LIN {X 0,Y 421.456,Z 405.097,A -85,B 0,C 180,E1 -19565.569,E2 -19565.569} C_VEL
LIN {X 0,Y 419.818,Z 402.472,A -85,B 0,C 180,E1 -19566.916,E2 -19566.916} C_VEL
LIN {X 0,Y 418.454,Z 400.452,A -85,B 0,C 180,E1 -19568.268,E2 -19568.268} C_VEL
LIN {X 0,Y 417.334,Z 399.088,A -85,B 0,C 180,E1 -19569.627,E2 -19569.627} C_VEL
LIN {X 0,Y 416.513,Z 398.311,A -85,B 0,C 180,E1 -19570.985,E2 -19570.985} C_VEL
LIN {X 0,Y 415.786,Z 398.064,A -85,B 0,C 180,E1 -19573.582,E2 -19573.582} C_VEL
LIN {X 0,Y 415.749,Z 398.727,A -85,B 0,C 180,E1 -19575.041,E2 -19575.041} C_VEL
LIN {X 0,Y 415.853,Z 399.961,A -85,B 0,C 180,E1 -19576.408,E2 -19576.408} C_VEL
LIN {X 0,Y 416.47,Z 403.077,A -85,B 0,C 180,E1 -19578.621,E2 -19578.621} C_VEL
LIN {X 0,Y 417.253,Z 406.927,A -85,B 0,C 180,E1 -19580.552,E2 -19580.552} C_VEL
LIN {X 0,Y 418.096,Z 411.291,A -85,B 0,C 180,E1 -19582.275,E2 -19582.275} C_VEL
LIN {X 0,Y 418.985,Z 417.288,A -85,B 0,C 180,E1 -19584.189,E2 -19584.189} C_VEL
LIN {X 0,Y 419.595,Z 423.229,A -85,B 0,C 180,E1 -19585.779,E2 -19585.779} C_VEL
LIN {X 0,Y 419.621,Z 425.888,A -85,B 0,C 180,E1 -19586.377,E2 -19586.377} C_VEL
LIN {X 0,Y 416.191,Z 439.912,A -85,B 0,C 180,E1 -19588.518,E2 -19588.518} C_VEL
LIN {X 0,Y 418.709,Z 457.984,A -85,B 0,C 180,E1 -19590.072,E2 -19590.072} C_VEL
LIN {X 0,Y 420.599,Z 474.74,A -85,B 0,C 180,E1 -19591.291,E2 -19591.291} C_VEL
LIN {X 0,Y 421.478,Z 486.634,A -85,B 0,C 180,E1 -19592.022,E2 -19592.022} C_VEL
LIN {X 0,Y 413.487,Z 565.78,A -85,B 0,C 180,E1 -19594.408,E2 -19594.408} C_VEL
LIN {X 0,Y 411.414,Z 585.881,A -85,B 0,C 180,E1 -19595.045,E2 -19595.045} C_VEL
LIN {X 0,Y 409.212,Z 601.626,A -85,B 0,C 180,E1 -19595.745,E2 -19595.745} C_VEL
LIN {X 0,Y 407.016,Z 615.192,A -85,B 0,C 180,E1 -19596.549,E2 -19596.549} C_VEL
LIN {X 0,Y 404.684,Z 627.697,A -85,B 0,C 180,E1 -19597.484,E2 -19597.484} C_VEL
LIN {X 0,Y 401.994,Z 640.642,A -85,B 0,C 180,E1 -19598.671,E2 -19598.671} C_VEL
LIN {X 0,Y 399.242,Z 652.442,A -85,B 0,C 180,E1 -19599.994,E2 -19599.994} C_VEL
LIN {X 0,Y 396.574,Z 663.167,A -85,B 0,C 180,E1 -19601.463,E2 -19601.463} C_VEL
LIN {X 0,Y 394.247,Z 672.105,A -85,B 0,C 180,E1 -19602.954,E2 -19602.954} C_VEL
LIN {X 0,Y 391.823,Z 680.778,A -85,B 0,C 180,E1 -19604.712,E2 -19604.712} C_VEL
LIN {X 0,Y 389.982,Z 687.808,A -85,B 0,C 180,E1 -19606.497,E2 -19606.497} C_VEL
LIN {X 0,Y 388.483,Z 692.746,A -85,B 0,C 180,E1 -19608.033,E2 -19608.033} C_VEL
LIN {X 0,Y 386.939,Z 697.849,A -85,B 0,C 180,E1 -19610.098,E2 -19610.098} C_VEL
LIN {X 0,Y 386.107,Z 700.668,A -85,B 0,C 180,E1 -19611.655,E2 -19611.655} C_VEL
LIN {X 0,Y 385.304,Z 703.116,A -85,B 0,C 180,E1 -19613.738,E2 -19613.738} C_VEL
LIN {X 0,Y 384.881,Z 704.141,A -85,B 0,C 180,E1 -19615.826,E2 -19615.826} C_VEL
LIN {X 0,Y 384.732,Z 703.738,A -85,B 0,C 180,E1 -19617.914,E2 -19617.914} C_VEL
LIN {X 0,Y 384.726,Z 701.892,A -85,B 0,C 180,E1 -19620,E2 -19620} C_VEL
LIN {X 0,Y 384.766,Z 698.539,A -85,B 0,C 180,E1 -19622.087,E2 -19622.087} C_VEL
LIN {X 0,Y 384.846,Z 693.513,A -85,B 0,C 180,E1 -19624.175,E2 -19624.175} C_VEL
LIN {X 0,Y 385.029,Z 687.035,A -85,B 0,C 180,E1 -19626.178,E2 -19626.178} C_VEL
LIN {X 0,Y 385.233,Z 680.259,A -85,B 0,C 180,E1 -19627.838,E2 -19627.838} C_VEL
LIN {X 0,Y 385.641,Z 672.491,A -85,B 0,C 180,E1 -19629.409,E2 -19629.409} C_VEL
LIN {X 0,Y 386.192,Z 663.141,A -85,B 0,C 180,E1 -19630.979,E2 -19630.979} C_VEL
LIN {X 0,Y 386.823,Z 653.048,A -85,B 0,C 180,E1 -19632.39,E2 -19632.39} C_VEL
LIN {X 0,Y 387.507,Z 641.531,A -85,B 0,C 180,E1 -19633.724,E2 -19633.724} C_VEL
LIN {X 0,Y 388.367,Z 627.771,A -85,B 0,C 180,E1 -19635.027,E2 -19635.027} C_VEL
LIN {X 0,Y 389.224,Z 614.122,A -85,B 0,C 180,E1 -19636.063,E2 -19636.063} C_VEL
LIN {X 0,Y 389.85,Z 599.788,A -85,B 0,C 180,E1 -19636.909,E2 -19636.909} C_VEL
LIN {X 0,Y 390.572,Z 584.437,A -85,B 0,C 180,E1 -19637.582,E2 -19637.582} C_VEL
LIN {X 0,Y 391.166,Z 565.272,A -85,B 0,C 180,E1 -19638.148,E2 -19638.148} C_VEL
LIN {X 0,Y 393.796,Z 473.423,A -85,B 0,C 180,E1 -19640.584,E2 -19640.584} C_VEL
LIN {X 0,Y 391.146,Z 442.771,A -85,B 0,C 180,E1 -19641.493,E2 -19641.493} C_VEL
LIN {X 0,Y 391.004,Z 439.485,A -85,B 0,C 180,E1 -19641.608,E2 -19641.608} C_VEL
LIN {X 0,Y 393.043,Z 410.801,A -85,B 0,C 180,E1 -19645.464,E2 -19645.464} C_VEL
LIN {X 0,Y 394.991,Z 385.613,A -85,B 0,C 180,E1 -19648.851,E2 -19648.851} C_VEL
LIN {X 0,Y 392.363,Z 372.738,A -85,B 0,C 180,E1 -19650.747,E2 -19650.747} C_VEL
LIN {X 0,Y 387.205,Z 349.81,A -85,B 0,C 180,E1 -19654.228,E2 -19654.228} C_VEL
LIN {X 0,Y 387.14,Z 349.817,A -85,B 0,C 180,E1 -19657.964,E2 -19657.964} C_VEL
LIN {X 0,Y 387.11,Z 349.82,A -85,B 0,C 180,E1 -19660.647,E2 -19660.647} C_VEL
LIN {X 0,Y 387.157,Z 349.814,A -85,B 0,C 180,E1 -19663.641,E2 -19663.641} C_VEL
LIN {X 0,Y 387.144,Z 349.816,A -85,B 0,C 180,E1 -19666.566,E2 -19666.566} C_VEL
LIN {X 0,Y 387.112,Z 349.817,A -85,B 0,C 180,E1 -19669.461,E2 -19669.461} C_VEL
LIN {X 0,Y 387.151,Z 349.818,A -85,B 0,C 180,E1 -19672.756,E2 -19672.756} C_VEL
LIN {X 0,Y 387.155,Z 349.814,A -85,B 0,C 180,E1 -19675.885,E2 -19675.885} C_VEL
LIN {X 0,Y 387.155,Z 349.811,A -85,B 0,C 180,E1 -19679.564,E2 -19679.564} C_VEL
LIN {X 0,Y 387.168,Z 349.814,A -85,B 0,C 180,E1 -19683.11,E2 -19683.11} C_VEL
LIN {X 0,Y 387.151,Z 349.815,A -85,B 0,C 180,E1 -19685.41,E2 -19685.41} C_VEL
LIN {X 0,Y 387.215,Z 349.808,A -85,B 0,C 180,E1 -19687.674,E2 -19687.674} C_VEL
LIN {X 0,Y 387.22,Z 349.81,A -85,B 0,C 180,E1 -19691.413,E2 -19691.413} C_VEL
LIN {X 0,Y 387.507,Z 351.104,A -85,B 0,C 180,E1 -19691.502,E2 -19691.502} C_VEL
LIN {X 0,Y 397.358,Z 374.738,A -85,B 0,C 180,E1 -19692.531,E2 -19692.531} C_VEL
LIN {X 0,Y 398.689,Z 378.334,A -85,B 0,C 180,E1 -19692.673,E2 -19692.673} C_VEL
LIN {X 0,Y 397.417,Z 458.29,A -85,B 0,C 180,E1 -19694.113,E2 -19694.113} C_VEL
LIN {X 0,Y 397.239,Z 474.684,A -85,B 0,C 180,E1 -19694.5,E2 -19694.5} C_VEL
LIN {X 0,Y 396.811,Z 488.678,A -85,B 0,C 180,E1 -19695.039,E2 -19695.039} C_VEL
LIN {X 0,Y 396.06,Z 502.62,A -85,B 0,C 180,E1 -19695.796,E2 -19695.796} C_VEL
LIN {X 0,Y 395.161,Z 515.096,A -85,B 0,C 180,E1 -19696.678,E2 -19696.678} C_VEL
LIN {X 0,Y 394.152,Z 527.624,A -85,B 0,C 180,E1 -19697.798,E2 -19697.798} C_VEL
LIN {X 0,Y 392.993,Z 539.27,A -85,B 0,C 180,E1 -19699.084,E2 -19699.084} C_VEL
LIN {X 0,Y 391.663,Z 549.672,A -85,B 0,C 180,E1 -19700.478,E2 -19700.478} C_VEL
LIN {X 0,Y 390.507,Z 559.045,A -85,B 0,C 180,E1 -19702.01,E2 -19702.01} C_VEL
LIN {X 0,Y 389.278,Z 568.029,A -85,B 0,C 180,E1 -19703.802,E2 -19703.802} C_VEL
LIN {X 0,Y 388.385,Z 574.313,A -85,B 0,C 180,E1 -19705.345,E2 -19705.345} C_VEL
LIN {X 0,Y 387.759,Z 579.507,A -85,B 0,C 180,E1 -19706.894,E2 -19706.894} C_VEL
LIN {X 0,Y 387.077,Z 584.999,A -85,B 0,C 180,E1 -19708.963,E2 -19708.963} C_VEL
LIN {X 0,Y 386.732,Z 588.97,A -85,B 0,C 180,E1 -19711.038,E2 -19711.038} C_VEL
LIN {X 0,Y 386.462,Z 591.568,A -85,B 0,C 180,E1 -19713.117,E2 -19713.117} C_VEL
LIN {X 0,Y 386.555,Z 592.824,A -85,B 0,C 180,E1 -19715.198,E2 -19715.198} C_VEL
LIN {X 0,Y 386.762,Z 592.797,A -85,B 0,C 180,E1 -19717.283,E2 -19717.283} C_VEL
LIN {X 0,Y 387.136,Z 591.478,A -85,B 0,C 180,E1 -19719.372,E2 -19719.372} C_VEL
LIN {X 0,Y 387.83,Z 588.815,A -85,B 0,C 180,E1 -19721.459,E2 -19721.459} C_VEL
LIN {X 0,Y 388.861,Z 584.721,A -85,B 0,C 180,E1 -19723.543,E2 -19723.543} C_VEL
LIN {X 0,Y 390.117,Z 579.079,A -85,B 0,C 180,E1 -19725.624,E2 -19725.624} C_VEL
LIN {X 0,Y 391.483,Z 572.687,A -85,B 0,C 180,E1 -19727.439,E2 -19727.439} C_VEL
LIN {X 0,Y 392.996,Z 565.164,A -85,B 0,C 180,E1 -19729.154,E2 -19729.154} C_VEL
LIN {X 0,Y 394.675,Z 556.34,A -85,B 0,C 180,E1 -19730.791,E2 -19730.791} C_VEL
LIN {X 0,Y 396.405,Z 546.158,A -85,B 0,C 180,E1 -19732.328,E2 -19732.328} C_VEL
LIN {X 0,Y 398.082,Z 534.772,A -85,B 0,C 180,E1 -19733.728,E2 -19733.728} C_VEL
LIN {X 0,Y 399.606,Z 523.258,A -85,B 0,C 180,E1 -19734.878,E2 -19734.878} C_VEL
LIN {X 0,Y 401.025,Z 510.621,A -85,B 0,C 180,E1 -19735.891,E2 -19735.891} C_VEL
LIN {X 0,Y 401.899,Z 498.61,A -85,B 0,C 180,E1 -19736.666,E2 -19736.666} C_VEL
LIN {X 0,Y 402.686,Z 484.904,A -85,B 0,C 180,E1 -19737.334,E2 -19737.334} C_VEL
LIN {X 0,Y 403.123,Z 470.306,A -85,B 0,C 180,E1 -19737.831,E2 -19737.831} C_VEL
LIN {X 0,Y 404.22,Z 419.999,A -85,B 0,C 180,E1 -19738.764,E2 -19738.764} C_VEL
LIN {X 0,Y 404.986,Z 387.088,A -85,B 0,C 180,E1 -19739.351,E2 -19739.351} C_VEL
LIN {X 0,Y 398.946,Z 373.795,A -85,B 0,C 180,E1 -19740.063,E2 -19740.063} C_VEL
LIN {X 0,Y 396.966,Z 370.73,A -85,B 0,C 180,E1 -19740.276,E2 -19740.276} C_VEL
LIN {X 0,Y 392.294,Z 367.019,A -85,B 0,C 180,E1 -19740.717,E2 -19740.717} C_VEL
LIN {X 0,Y 387.387,Z 363.5,A -85,B 0,C 180,E1 -19741.186,E2 -19741.186} C_VEL
LIN {X 0,Y 385.044,Z 360.686,A -85,B 0,C 180,E1 -19741.438,E2 -19741.438} C_VEL
LIN {X 0,Y 380.323,Z 351.887,A -85,B 0,C 180,E1 -19742.026,E2 -19742.026} C_VEL
LIN {X 0,Y 380.053,Z 350.704,A -85,B 0,C 180,E1 -19742.097,E2 -19742.097} C_VEL
LIN {X 0,Y 380.058,Z 350.7,A -85,B 0,C 180,E1 -19745.814,E2 -19745.814} C_VEL
LIN {X 0,Y 380.075,Z 350.7,A -85,B 0,C 180,E1 -19749.283,E2 -19749.283} C_VEL
LIN {X 0,Y 380.017,Z 350.708,A -85,B 0,C 180,E1 -19752.999,E2 -19752.999} C_VEL
LIN {X 0,Y 380.068,Z 350.701,A -85,B 0,C 180,E1 -19755.952,E2 -19755.952} C_VEL
LIN {X 0,Y 380.06,Z 350.703,A -85,B 0,C 180,E1 -19759.83,E2 -19759.83} C_VEL
LIN {X 0,Y 380.092,Z 350.659,A -85,B 0,C 180,E1 -19762.545,E2 -19762.545} C_VEL
LIN {X 0,Y 380.055,Z 350.691,A -85,B 0,C 180,E1 -19766.033,E2 -19766.033} C_VEL
LIN {X 0,Y 380.061,Z 350.69,A -85,B 0,C 180,E1 -19768.933,E2 -19768.933} C_VEL
LIN {X 0,Y 380.138,Z 350.686,A -85,B 0,C 180,E1 -19772.57,E2 -19772.57} C_VEL
LIN {X 0,Y 380.083,Z 350.699,A -85,B 0,C 180,E1 -19776.081,E2 -19776.081} C_VEL
LIN {X 0,Y 380.116,Z 350.684,A -85,B 0,C 180,E1 -19778.196,E2 -19778.196} C_VEL
LIN {X 0,Y 386.254,Z 373.597,A -85,B 0,C 180,E1 -19779.015,E2 -19779.015} C_VEL
LIN {X 0,Y 383.978,Z 466.755,A -85,B 0,C 180,E1 -19781.515,E2 -19781.515} C_VEL
LIN {X 0,Y 383.681,Z 482.142,A -85,B 0,C 180,E1 -19782.125,E2 -19782.125} C_VEL
LIN {X 0,Y 383.162,Z 496.898,A -85,B 0,C 180,E1 -19782.924,E2 -19782.924} C_VEL
LIN {X 0,Y 382.541,Z 511.111,A -85,B 0,C 180,E1 -19783.922,E2 -19783.922} C_VEL
LIN {X 0,Y 381.806,Z 524.693,A -85,B 0,C 180,E1 -19785.117,E2 -19785.117} C_VEL
LIN {X 0,Y 381.211,Z 537.097,A -85,B 0,C 180,E1 -19786.451,E2 -19786.451} C_VEL
LIN {X 0,Y 380.611,Z 549.201,A -85,B 0,C 180,E1 -19788.051,E2 -19788.051} C_VEL
LIN {X 0,Y 380.015,Z 559.208,A -85,B 0,C 180,E1 -19789.647,E2 -19789.647} C_VEL
LIN {X 0,Y 379.592,Z 567.569,A -85,B 0,C 180,E1 -19791.243,E2 -19791.243} C_VEL
LIN {X 0,Y 379.244,Z 575.608,A -85,B 0,C 180,E1 -19793.105,E2 -19793.105} C_VEL
LIN {X 0,Y 379.12,Z 581.229,A -85,B 0,C 180,E1 -19794.699,E2 -19794.699} C_VEL
LIN {X 0,Y 379.161,Z 586.5,A -85,B 0,C 180,E1 -19796.568,E2 -19796.568} C_VEL
LIN {X 0,Y 379.226,Z 589.413,A -85,B 0,C 180,E1 -19797.883,E2 -19797.883} C_VEL
LIN {X 0,Y 379.447,Z 592.933,A -85,B 0,C 180,E1 -19800,E2 -19800} C_VEL
LIN {X 0,Y 379.774,Z 594.135,A -85,B 0,C 180,E1 -19801.057,E2 -19801.057} C_VEL
LIN {X 0,Y 380.467,Z 595.445,A -85,B 0,C 180,E1 -19803.166,E2 -19803.166} C_VEL
LIN {X 0,Y 381.466,Z 595.301,A -85,B 0,C 180,E1 -19805.267,E2 -19805.267} C_VEL
LIN {X 0,Y 382.746,Z 593.753,A -85,B 0,C 180,E1 -19807.36,E2 -19807.36} C_VEL
LIN {X 0,Y 384.467,Z 590.727,A -85,B 0,C 180,E1 -19809.437,E2 -19809.437} C_VEL
LIN {X 0,Y 386.204,Z 587.375,A -85,B 0,C 180,E1 -19810.978,E2 -19810.978} C_VEL
LIN {X 0,Y 388.299,Z 582.106,A -85,B 0,C 180,E1 -19812.846,E2 -19812.846} C_VEL
LIN {X 0,Y 390.456,Z 575.96,A -85,B 0,C 180,E1 -19814.545,E2 -19814.545} C_VEL
LIN {X 0,Y 393.004,Z 567.926,A -85,B 0,C 180,E1 -19816.302,E2 -19816.302} C_VEL
LIN {X 0,Y 395.325,Z 559.584,A -85,B 0,C 180,E1 -19817.796,E2 -19817.796} C_VEL
LIN {X 0,Y 397.897,Z 549.476,A -85,B 0,C 180,E1 -19819.273,E2 -19819.273} C_VEL
LIN {X 0,Y 400.462,Z 538.325,A -85,B 0,C 180,E1 -19820.61,E2 -19820.61} C_VEL
LIN {X 0,Y 402.689,Z 527.29,A -85,B 0,C 180,E1 -19821.692,E2 -19821.692} C_VEL
LIN {X 0,Y 404.918,Z 513.604,A -85,B 0,C 180,E1 -19822.797,E2 -19822.797} C_VEL
LIN {X 0,Y 406.637,Z 500.309,A -85,B 0,C 180,E1 -19823.657,E2 -19823.657} C_VEL
LIN {X 0,Y 408.023,Z 486.215,A -85,B 0,C 180,E1 -19824.368,E2 -19824.368} C_VEL
LIN {X 0,Y 409.477,Z 466.445,A -85,B 0,C 180,E1 -19825.081,E2 -19825.081} C_VEL
LIN {X 0,Y 415.8,Z 403.546,A -85,B 0,C 180,E1 -19827.01,E2 -19827.01} C_VEL
LIN {X 0,Y 411.197,Z 394.797,A -85,B 0,C 180,E1 -19828.316,E2 -19828.316} C_VEL
LIN {X 0,Y 407.426,Z 388.228,A -85,B 0,C 180,E1 -19829.488,E2 -19829.488} C_VEL
LIN {X 0,Y 404.57,Z 383.673,A -85,B 0,C 180,E1 -19830.432,E2 -19830.432} C_VEL
LIN {X 0,Y 402.64,Z 380.748,A -85,B 0,C 180,E1 -19831.1,E2 -19831.1} C_VEL
LIN {X 0,Y 400.122,Z 376.96,A -85,B 0,C 180,E1 -19832.072,E2 -19832.072} C_VEL
LIN {X 0,Y 397.798,Z 373.541,A -85,B 0,C 180,E1 -19833.046,E2 -19833.046} C_VEL
LIN {X 0,Y 396.698,Z 372.184,A -85,B 0,C 180,E1 -19833.536,E2 -19833.536} C_VEL
LIN {X 0,Y 394.522,Z 369.343,A -85,B 0,C 180,E1 -19834.557,E2 -19834.557} C_VEL
LIN {X 0,Y 393.669,Z 367.713,A -85,B 0,C 180,E1 -19835.068,E2 -19835.068} C_VEL
LIN {X 0,Y 391.139,Z 365.315,A -85,B 0,C 180,E1 -19836.487,E2 -19836.487} C_VEL
LIN {X 0,Y 389.358,Z 362.272,A -85,B 0,C 180,E1 -19837.967,E2 -19837.967} C_VEL
LIN {X 0,Y 386.416,Z 360.095,A -85,B 0,C 180,E1 -19841.249,E2 -19841.249} C_VEL
LIN {X 0,Y 386.073,Z 359.582,A -85,B 0,C 180,E1 -19843.584,E2 -19843.584} C_VEL
LIN {X 0,Y 386.641,Z 360.248,A -85,B 0,C 180,E1 -19845.691,E2 -19845.691} C_VEL
LIN {X 0,Y 389.268,Z 362.251,A -85,B 0,C 180,E1 -19848.748,E2 -19848.748} C_VEL
LIN {X 0,Y 389.637,Z 362.726,A -85,B 0,C 180,E1 -19849.077,E2 -19849.077} C_VEL
LIN {X 0,Y 391.078,Z 365.663,A -85,B 0,C 180,E1 -19850.368,E2 -19850.368} C_VEL
LIN {X 0,Y 393.603,Z 368.05,A -85,B 0,C 180,E1 -19851.849,E2 -19851.849} C_VEL
LIN {X 0,Y 395.337,Z 371.427,A -85,B 0,C 180,E1 -19852.9,E2 -19852.9} C_VEL
LIN {X 0,Y 398.706,Z 382.971,A -85,B 0,C 180,E1 -19855.006,E2 -19855.006} C_VEL
LIN {X 0,Y 403.21,Z 398.657,A -85,B 0,C 180,E1 -19857.253,E2 -19857.253} C_VEL
LIN {X 0,Y 404.435,Z 403.83,A -85,B 0,C 180,E1 -19857.845,E2 -19857.845} C_VEL
LIN {X 0,Y 406.35,Z 425.682,A -85,B 0,C 180,E1 -19859.485,E2 -19859.485} C_VEL
LIN {X 0,Y 408.013,Z 448.682,A -85,B 0,C 180,E1 -19860.97,E2 -19860.97} C_VEL
LIN {X 0,Y 408.777,Z 467.334,A -85,B 0,C 180,E1 -19861.99,E2 -19861.99} C_VEL
LIN {X 0,Y 408.658,Z 484.147,A -85,B 0,C 180,E1 -19862.744,E2 -19862.744} C_VEL
LIN {X 0,Y 402.992,Z 544.44,A -85,B 0,C 180,E1 -19864.589,E2 -19864.589} C_VEL
LIN {X 0,Y 400.692,Z 560.631,A -85,B 0,C 180,E1 -19865.263,E2 -19865.263} C_VEL
LIN {X 0,Y 397.939,Z 576.004,A -85,B 0,C 180,E1 -19866.119,E2 -19866.119} C_VEL
LIN {X 0,Y 394.826,Z 590.77,A -85,B 0,C 180,E1 -19867.165,E2 -19867.165} C_VEL
LIN {X 0,Y 392.079,Z 602.814,A -85,B 0,C 180,E1 -19868.241,E2 -19868.241} C_VEL
LIN {X 0,Y 388.977,Z 615.663,A -85,B 0,C 180,E1 -19869.662,E2 -19869.662} C_VEL
LIN {X 0,Y 386.213,Z 627.166,A -85,B 0,C 180,E1 -19871.221,E2 -19871.221} C_VEL
LIN {X 0,Y 383.863,Z 636.49,A -85,B 0,C 180,E1 -19872.751,E2 -19872.751} C_VEL
LIN {X 0,Y 381.714,Z 645.61,A -85,B 0,C 180,E1 -19874.569,E2 -19874.569} C_VEL
LIN {X 0,Y 380.437,Z 652.119,A -85,B 0,C 180,E1 -19876.152,E2 -19876.152} C_VEL
LIN {X 0,Y 379.291,Z 658.883,A -85,B 0,C 180,E1 -19878.17,E2 -19878.17} C_VEL
LIN {X 0,Y 379.1,Z 660.118,A -85,B 0,C 180,E1 -19878.505,E2 -19878.505} C_VEL
LIN {X 0,Y 378.606,Z 670.59,A -85,B 0,C 180,E1 -19880.146,E2 -19880.146} C_VEL
LIN {X 0,Y 378.182,Z 679.031,A -85,B 0,C 180,E1 -19881.747,E2 -19881.747} C_VEL
LIN {X 0,Y 378.032,Z 686.038,A -85,B 0,C 180,E1 -19883.35,E2 -19883.35} C_VEL
LIN {X 0,Y 377.878,Z 692.63,A -85,B 0,C 180,E1 -19885.215,E2 -19885.215} C_VEL
LIN {X 0,Y 377.769,Z 697.072,A -85,B 0,C 180,E1 -19886.811,E2 -19886.811} C_VEL
LIN {X 0,Y 377.747,Z 700.554,A -85,B 0,C 180,E1 -19888.406,E2 -19888.406} C_VEL
LIN {X 0,Y 377.763,Z 703.112,A -85,B 0,C 180,E1 -19890,E2 -19890} C_VEL
LIN {X 0,Y 377.697,Z 705.177,A -85,B 0,C 180,E1 -19892.125,E2 -19892.125} C_VEL
LIN {X 0,Y 377.805,Z 705.754,A -85,B 0,C 180,E1 -19894.253,E2 -19894.253} C_VEL
LIN {X 0,Y 378.224,Z 704.888,A -85,B 0,C 180,E1 -19896.38,E2 -19896.38} C_VEL
LIN {X 0,Y 378.953,Z 702.596,A -85,B 0,C 180,E1 -19898.503,E2 -19898.503} C_VEL
LIN {X 0,Y 380.08,Z 698.85,A -85,B 0,C 180,E1 -19900.62,E2 -19900.62} C_VEL
LIN {X 0,Y 381.989,Z 693.512,A -85,B 0,C 180,E1 -19902.711,E2 -19902.711} C_VEL
LIN {X 0,Y 383.71,Z 687.091,A -85,B 0,C 180,E1 -19904.65,E2 -19904.65} C_VEL
LIN {X 0,Y 385.876,Z 679.96,A -85,B 0,C 180,E1 -19906.341,E2 -19906.341} C_VEL
LIN {X 0,Y 388.164,Z 672.161,A -85,B 0,C 180,E1 -19907.864,E2 -19907.864} C_VEL
LIN {X 0,Y 390.676,Z 662.882,A -85,B 0,C 180,E1 -19909.371,E2 -19909.371} C_VEL
LIN {X 0,Y 393.55,Z 651.743,A -85,B 0,C 180,E1 -19910.852,E2 -19910.852} C_VEL
LIN {X 0,Y 396.465,Z 639.495,A -85,B 0,C 180,E1 -19912.187,E2 -19912.187} C_VEL
LIN {X 0,Y 399.052,Z 627.406,A -85,B 0,C 180,E1 -19913.262,E2 -19913.262} C_VEL
LIN {X 0,Y 401.633,Z 614.287,A -85,B 0,C 180,E1 -19914.195,E2 -19914.195} C_VEL
LIN {X 0,Y 403.663,Z 602.24,A -85,B 0,C 180,E1 -19914.884,E2 -19914.884} C_VEL
LIN {X 0,Y 405.985,Z 585.949,A -85,B 0,C 180,E1 -19915.586,E2 -19915.586} C_VEL
LIN {X 0,Y 416.69,Z 486.417,A -85,B 0,C 180,E1 -19918.703,E2 -19918.703} C_VEL
LIN {X 0,Y 416.964,Z 474.884,A -85,B 0,C 180,E1 -19919.257,E2 -19919.257} C_VEL
LIN {X 0,Y 416.688,Z 456.276,A -85,B 0,C 180,E1 -19920.337,E2 -19920.337} C_VEL
LIN {X 0,Y 415.676,Z 437.783,A -85,B 0,C 180,E1 -19921.668,E2 -19921.668} C_VEL
LIN {X 0,Y 417.96,Z 421.947,A -85,B 0,C 180,E1 -19923.431,E2 -19923.431} C_VEL
LIN {X 0,Y 418.953,Z 416.867,A -85,B 0,C 180,E1 -19924.036,E2 -19924.036} C_VEL
LIN {X 0,Y 419.108,Z 415.056,A -85,B 0,C 180,E1 -19924.324,E2 -19924.324} C_VEL
LIN {X 0,Y 418.985,Z 413.617,A -85,B 0,C 180,E1 -19924.639,E2 -19924.639} C_VEL
LIN {X 0,Y 416.871,Z 409.812,A -85,B 0,C 180,E1 -19926.243,E2 -19926.243} C_VEL
LIN {X 0,Y 415.364,Z 407.52,A -85,B 0,C 180,E1 -19927.573,E2 -19927.573} C_VEL
LIN {X 0,Y 414.11,Z 405.813,A -85,B 0,C 180,E1 -19928.916,E2 -19928.916} C_VEL
LIN {X 0,Y 413.094,Z 404.682,A -85,B 0,C 180,E1 -19930.269,E2 -19930.269} C_VEL
LIN {X 0,Y 412.342,Z 404.054,A -85,B 0,C 180,E1 -19931.632,E2 -19931.632} C_VEL
LIN {X 0,Y 411.899,Z 403.923,A -85,B 0,C 180,E1 -19933.011,E2 -19933.011} C_VEL
LIN {X 0,Y 411.735,Z 404.274,A -85,B 0,C 180,E1 -19934.398,E2 -19934.398} C_VEL
LIN {X 0,Y 411.719,Z 405.22,A -85,B 0,C 180,E1 -19935.772,E2 -19935.772} C_VEL
LIN {X 0,Y 411.857,Z 406.677,A -85,B 0,C 180,E1 -19937.135,E2 -19937.135} C_VEL
LIN {X 0,Y 412.377,Z 409.84,A -85,B 0,C 180,E1 -19939.173,E2 -19939.173} C_VEL
LIN {X 0,Y 413.137,Z 414.328,A -85,B 0,C 180,E1 -19941.251,E2 -19941.251} C_VEL
LIN {X 0,Y 413.848,Z 419.251,A -85,B 0,C 180,E1 -19943.047,E2 -19943.047} C_VEL
LIN {X 0,Y 414.517,Z 426.503,A -85,B 0,C 180,E1 -19945.155,E2 -19945.155} C_VEL
LIN {X 0,Y 414.578,Z 429.416,A -85,B 0,C 180,E1 -19945.881,E2 -19945.881} C_VEL
LIN {X 0,Y 411.884,Z 439.997,A -85,B 0,C 180,E1 -19947.52,E2 -19947.52} C_VEL
LIN {X 0,Y 414.02,Z 456.862,A -85,B 0,C 180,E1 -19949.063,E2 -19949.063} C_VEL
LIN {X 0,Y 415.934,Z 475.046,A -85,B 0,C 180,E1 -19950.468,E2 -19950.468} C_VEL
LIN {X 0,Y 416.819,Z 488.022,A -85,B 0,C 180,E1 -19951.307,E2 -19951.307} C_VEL
LIN {X 0,Y 408.399,Z 566.582,A -85,B 0,C 180,E1 -19953.723,E2 -19953.723} C_VEL
LIN {X 0,Y 406.257,Z 586.18,A -85,B 0,C 180,E1 -19954.364,E2 -19954.364} C_VEL
LIN {X 0,Y 403.951,Z 601.751,A -85,B 0,C 180,E1 -19955.066,E2 -19955.066} C_VEL
LIN {X 0,Y 401.488,Z 616.015,A -85,B 0,C 180,E1 -19955.933,E2 -19955.933} C_VEL
LIN {X 0,Y 398.72,Z 629.748,A -85,B 0,C 180,E1 -19956.991,E2 -19956.991} C_VEL
LIN {X 0,Y 395.942,Z 642.288,A -85,B 0,C 180,E1 -19958.192,E2 -19958.192} C_VEL
LIN {X 0,Y 393.346,Z 652.804,A -85,B 0,C 180,E1 -19959.409,E2 -19959.409} C_VEL
LIN {X 0,Y 390.494,Z 663.417,A -85,B 0,C 180,E1 -19960.892,E2 -19960.892} C_VEL
LIN {X 0,Y 387.632,Z 673.633,A -85,B 0,C 180,E1 -19962.654,E2 -19962.654} C_VEL
LIN {X 0,Y 385.096,Z 682.024,A -85,B 0,C 180,E1 -19964.438,E2 -19964.438} C_VEL
LIN {X 0,Y 383.16,Z 688.823,A -85,B 0,C 180,E1 -19966.252,E2 -19966.252} C_VEL
LIN {X 0,Y 381.604,Z 693.54,A -85,B 0,C 180,E1 -19967.814,E2 -19967.814} C_VEL
LIN {X 0,Y 379.96,Z 698.448,A -85,B 0,C 180,E1 -19969.914,E2 -19969.914} C_VEL
LIN {X 0,Y 379.1,Z 701.077,A -85,B 0,C 180,E1 -19971.5,E2 -19971.5} C_VEL
LIN {X 0,Y 378.254,Z 703.348,A -85,B 0,C 180,E1 -19973.621,E2 -19973.621} C_VEL
LIN {X 0,Y 377.8,Z 704.201,A -85,B 0,C 180,E1 -19975.747,E2 -19975.747} C_VEL
LIN {X 0,Y 377.647,Z 703.63,A -85,B 0,C 180,E1 -19977.874,E2 -19977.874} C_VEL
LIN {X 0,Y 377.657,Z 701.591,A -85,B 0,C 180,E1 -19980,E2 -19980} C_VEL
LIN {X 0,Y 377.704,Z 698.015,A -85,B 0,C 180,E1 -19982.126,E2 -19982.126} C_VEL
LIN {X 0,Y 377.794,Z 692.818,A -85,B 0,C 180,E1 -19984.253,E2 -19984.253} C_VEL
LIN {X 0,Y 377.954,Z 686.459,A -85,B 0,C 180,E1 -19986.204,E2 -19986.204} C_VEL
LIN {X 0,Y 378.181,Z 679.159,A -85,B 0,C 180,E1 -19987.985,E2 -19987.985} C_VEL
LIN {X 0,Y 378.619,Z 671.149,A -85,B 0,C 180,E1 -19989.585,E2 -19989.585} C_VEL
LIN {X 0,Y 379.129,Z 661.464,A -85,B 0,C 180,E1 -19991.186,E2 -19991.186} C_VEL
LIN {X 0,Y 379.911,Z 649.755,A -85,B 0,C 180,E1 -19992.783,E2 -19992.783} C_VEL
LIN {X 0,Y 380.591,Z 637.89,A -85,B 0,C 180,E1 -19994.114,E2 -19994.114} C_VEL
LIN {X 0,Y 381.473,Z 624.89,A -85,B 0,C 180,E1 -19995.305,E2 -19995.305} C_VEL
LIN {X 0,Y 382.333,Z 610.405,A -85,B 0,C 180,E1 -19996.36,E2 -19996.36} C_VEL
LIN {X 0,Y 382.983,Z 596.436,A -85,B 0,C 180,E1 -19997.153,E2 -19997.153} C_VEL
LIN {X 0,Y 383.607,Z 581.425,A -85,B 0,C 180,E1 -19997.775,E2 -19997.775} C_VEL
LIN {X 0,Y 386.811,Z 473.812,A -85,B 0,C 180,E1 -20000.747,E2 -20000.747} C_VEL
LIN {X 0,Y 384.17,Z 443.194,A -85,B 0,C 180,E1 -20001.677,E2 -20001.677} C_VEL
LIN {X 0,Y 384.034,Z 439.615,A -85,B 0,C 180,E1 -20001.791,E2 -20001.791} C_VEL
LIN {X 0,Y 386.09,Z 411.203,A -85,B 0,C 180,E1 -20005.653,E2 -20005.653} C_VEL
LIN {X 0,Y 387.994,Z 386.44,A -85,B 0,C 180,E1 -20009.024,E2 -20009.024} C_VEL
LIN {X 0,Y 384.539,Z 370.129,A -85,B 0,C 180,E1 -20011.471,E2 -20011.471} C_VEL
LIN {X 0,Y 380.135,Z 350.691,A -85,B 0,C 180,E1 -20014.478,E2 -20014.478} C_VEL
LIN {X 0,Y 380.094,Z 350.697,A -85,B 0,C 180,E1 -20017.588,E2 -20017.588} C_VEL
LIN {X 0,Y 380.052,Z 350.7,A -85,B 0,C 180,E1 -20020.919,E2 -20020.919} C_VEL
LIN {X 0,Y 380.122,Z 350.691,A -85,B 0,C 180,E1 -20024.445,E2 -20024.445} C_VEL
LIN {X 0,Y 380.088,Z 350.696,A -85,B 0,C 180,E1 -20027.489,E2 -20027.489} C_VEL
LIN {X 0,Y 380.083,Z 350.697,A -85,B 0,C 180,E1 -20031.202,E2 -20031.202} C_VEL
LIN {X 0,Y 380.104,Z 350.691,A -85,B 0,C 180,E1 -20034.177,E2 -20034.177} C_VEL
LIN {X 0,Y 380.099,Z 350.687,A -85,B 0,C 180,E1 -20037.696,E2 -20037.696} C_VEL
LIN {X 0,Y 380.137,Z 350.688,A -85,B 0,C 180,E1 -20040.165,E2 -20040.165} C_VEL
LIN {X 0,Y 380.116,Z 350.692,A -85,B 0,C 180,E1 -20043.753,E2 -20043.753} C_VEL
LIN {X 0,Y 380.141,Z 350.689,A -85,B 0,C 180,E1 -20047.236,E2 -20047.236} C_VEL
LIN {X 0,Y 380.175,Z 350.688,A -85,B 0,C 180,E1 -20050.998,E2 -20050.998} C_VEL
LIN {X 0,Y 380.548,Z 352.2,A -85,B 0,C 180,E1 -20051.096,E2 -20051.096} C_VEL
LIN {X 0,Y 390.867,Z 376.775,A -85,B 0,C 180,E1 -20052.201,E2 -20052.201} C_VEL
LIN {X 0,Y 392.163,Z 380.716,A -85,B 0,C 180,E1 -20052.351,E2 -20052.351} C_VEL
LIN {X 0,Y 390.737,Z 454.982,A -85,B 0,C 180,E1 -20053.701,E2 -20053.701} C_VEL
LIN {X 0,Y 390.616,Z 472.829,A -85,B 0,C 180,E1 -20054.096,E2 -20054.096} C_VEL
LIN {X 0,Y 390.229,Z 486.981,A -85,B 0,C 180,E1 -20054.614,E2 -20054.614} C_VEL
LIN {X 0,Y 389.484,Z 501.168,A -85,B 0,C 180,E1 -20055.351,E2 -20055.351} C_VEL
LIN {X 0,Y 388.565,Z 513.313,A -85,B 0,C 180,E1 -20056.181,E2 -20056.181} C_VEL
LIN {X 0,Y 387.652,Z 525.242,A -85,B 0,C 180,E1 -20057.212,E2 -20057.212} C_VEL
LIN {X 0,Y 386.487,Z 537.318,A -85,B 0,C 180,E1 -20058.501,E2 -20058.501} C_VEL
LIN {X 0,Y 385.218,Z 547.296,A -85,B 0,C 180,E1 -20059.788,E2 -20059.788} C_VEL
LIN {X 0,Y 383.908,Z 557.203,A -85,B 0,C 180,E1 -20061.343,E2 -20061.343} C_VEL
LIN {X 0,Y 382.792,Z 565.433,A -85,B 0,C 180,E1 -20062.905,E2 -20062.905} C_VEL
LIN {X 0,Y 381.715,Z 573.297,A -85,B 0,C 180,E1 -20064.736,E2 -20064.736} C_VEL
LIN {X 0,Y 380.89,Z 578.86,A -85,B 0,C 180,E1 -20066.31,E2 -20066.31} C_VEL
LIN {X 0,Y 380.197,Z 584.671,A -85,B 0,C 180,E1 -20068.417,E2 -20068.417} C_VEL
LIN {X 0,Y 379.792,Z 588.043,A -85,B 0,C 180,E1 -20070,E2 -20070} C_VEL
LIN {X 0,Y 379.555,Z 591.268,A -85,B 0,C 180,E1 -20072.115,E2 -20072.115} C_VEL
LIN {X 0,Y 379.409,Z 593.155,A -85,B 0,C 180,E1 -20074.235,E2 -20074.235} C_VEL
LIN {X 0,Y 379.586,Z 593.734,A -85,B 0,C 180,E1 -20076.357,E2 -20076.357} C_VEL
LIN {X 0,Y 379.927,Z 593.028,A -85,B 0,C 180,E1 -20078.482,E2 -20078.482} C_VEL
LIN {X 0,Y 380.414,Z 591.019,A -85,B 0,C 180,E1 -20080.61,E2 -20080.61} C_VEL
LIN {X 0,Y 381.416,Z 587.611,A -85,B 0,C 180,E1 -20082.731,E2 -20082.731} C_VEL
LIN {X 0,Y 382.565,Z 582.73,A -85,B 0,C 180,E1 -20084.853,E2 -20084.853} C_VEL
LIN {X 0,Y 384.062,Z 576.204,A -85,B 0,C 180,E1 -20086.966,E2 -20086.966} C_VEL
LIN {X 0,Y 385.641,Z 568.881,A -85,B 0,C 180,E1 -20088.808,E2 -20088.808} C_VEL
LIN {X 0,Y 387.158,Z 561.209,A -85,B 0,C 180,E1 -20090.382,E2 -20090.382} C_VEL
LIN {X 0,Y 388.886,Z 551.921,A -85,B 0,C 180,E1 -20091.947,E2 -20091.947} C_VEL
LIN {X 0,Y 390.73,Z 541.087,A -85,B 0,C 180,E1 -20093.434,E2 -20093.434} C_VEL
LIN {X 0,Y 392.263,Z 530.16,A -85,B 0,C 180,E1 -20094.671,E2 -20094.671} C_VEL
LIN {X 0,Y 393.926,Z 517.42,A -85,B 0,C 180,E1 -20095.826,E2 -20095.826} C_VEL
LIN {X 0,Y 395.036,Z 504.923,A -85,B 0,C 180,E1 -20096.739,E2 -20096.739} C_VEL
LIN {X 0,Y 395.958,Z 491.632,A -85,B 0,C 180,E1 -20097.488,E2 -20097.488} C_VEL
LIN {X 0,Y 396.642,Z 477.251,A -85,B 0,C 180,E1 -20098.072,E2 -20098.072} C_VEL
LIN {X 0,Y 396.908,Z 463.477,A -85,B 0,C 180,E1 -20098.431,E2 -20098.431} C_VEL
LIN {X 0,Y 398.591,Z 388.889,A -85,B 0,C 180,E1 -20099.788,E2 -20099.788} C_VEL
LIN {X 0,Y 389.633,Z 369.697,A -85,B 0,C 180,E1 -20100.875,E2 -20100.875} C_VEL
LIN {X 0,Y 385.044,Z 360.686,A -85,B 0,C 180,E1 -20101.438,E2 -20101.438} C_VEL
LIN {X 0,Y 383.498,Z 359.091,A -85,B 0,C 180,E1 -20101.602,E2 -20101.602} C_VEL
LIN {X 0,Y 380.11,Z 357.681,A -85,B 0,C 180,E1 -20101.92,E2 -20101.92} C_VEL
LIN {X 0,Y 375.516,Z 355.988,A -85,B 0,C 180,E1 -20102.359,E2 -20102.359} C_VEL
LIN {X 0,Y 374.624,Z 355.277,A -85,B 0,C 180,E1 -20102.454,E2 -20102.454} C_VEL
LIN {X 0,Y 373.264,Z 352.794,A -85,B 0,C 180,E1 -20102.631,E2 -20102.631} C_VEL
LIN {X 0,Y 372.983,Z 351.581,A -85,B 0,C 180,E1 -20102.71,E2 -20102.71} C_VEL
LIN {X 0,Y 373.032,Z 351.576,A -85,B 0,C 180,E1 -20106.155,E2 -20106.155} C_VEL
LIN {X 0,Y 373.014,Z 351.578,A -85,B 0,C 180,E1 -20109.677,E2 -20109.677} C_VEL
LIN {X 0,Y 372.976,Z 351.586,A -85,B 0,C 180,E1 -20112.91,E2 -20112.91} C_VEL
LIN {X 0,Y 373.027,Z 351.579,A -85,B 0,C 180,E1 -20115.991,E2 -20115.991} C_VEL
LIN {X 0,Y 372.988,Z 351.579,A -85,B 0,C 180,E1 -20118.907,E2 -20118.907} C_VEL
LIN {X 0,Y 373.011,Z 351.548,A -85,B 0,C 180,E1 -20122.063,E2 -20122.063} C_VEL
LIN {X 0,Y 372.999,Z 351.545,A -85,B 0,C 180,E1 -20124.398,E2 -20124.398} C_VEL
LIN {X 0,Y 373,Z 351.579,A -85,B 0,C 180,E1 -20127.677,E2 -20127.677} C_VEL
LIN {X 0,Y 373.023,Z 351.572,A -85,B 0,C 180,E1 -20130.776,E2 -20130.776} C_VEL
LIN {X 0,Y 373.096,Z 351.556,A -85,B 0,C 180,E1 -20134.418,E2 -20134.418} C_VEL
LIN {X 0,Y 373.095,Z 351.56,A -85,B 0,C 180,E1 -20138.053,E2 -20138.053} C_VEL
LIN {X 0,Y 379.227,Z 374.481,A -85,B 0,C 180,E1 -20138.869,E2 -20138.869} C_VEL
LIN {X 0,Y 376.874,Z 469.113,A -85,B 0,C 180,E1 -20141.489,E2 -20141.489} C_VEL
LIN {X 0,Y 376.585,Z 484.343,A -85,B 0,C 180,E1 -20142.127,E2 -20142.127} C_VEL
LIN {X 0,Y 376.082,Z 497.622,A -85,B 0,C 180,E1 -20142.872,E2 -20142.872} C_VEL
LIN {X 0,Y 375.437,Z 511.808,A -85,B 0,C 180,E1 -20143.887,E2 -20143.887} C_VEL
LIN {X 0,Y 374.733,Z 525.391,A -85,B 0,C 180,E1 -20145.107,E2 -20145.107} C_VEL
LIN {X 0,Y 374.08,Z 538.243,A -85,B 0,C 180,E1 -20146.519,E2 -20146.519} C_VEL
LIN {X 0,Y 373.48,Z 549.937,A -85,B 0,C 180,E1 -20148.094,E2 -20148.094} C_VEL
LIN {X 0,Y 372.897,Z 559.986,A -85,B 0,C 180,E1 -20149.72,E2 -20149.72} C_VEL
LIN {X 0,Y 372.479,Z 568.364,A -85,B 0,C 180,E1 -20151.347,E2 -20151.347} C_VEL
LIN {X 0,Y 372.141,Z 576.419,A -85,B 0,C 180,E1 -20153.244,E2 -20153.244} C_VEL
LIN {X 0,Y 372.041,Z 582.868,A -85,B 0,C 180,E1 -20155.14,E2 -20155.14} C_VEL
LIN {X 0,Y 372.139,Z 588.579,A -85,B 0,C 180,E1 -20157.303,E2 -20157.303} C_VEL
LIN {X 0,Y 372.238,Z 591.799,A -85,B 0,C 180,E1 -20158.922,E2 -20158.922} C_VEL
LIN {X 0,Y 372.717,Z 594.765,A -85,B 0,C 180,E1 -20161.077,E2 -20161.077} C_VEL
LIN {X 0,Y 373.435,Z 596.304,A -85,B 0,C 180,E1 -20163.225,E2 -20163.225} C_VEL
LIN {X 0,Y 374.491,Z 596.408,A -85,B 0,C 180,E1 -20165.366,E2 -20165.366} C_VEL
LIN {X 0,Y 375.826,Z 595.055,A -85,B 0,C 180,E1 -20167.496,E2 -20167.496} C_VEL
LIN {X 0,Y 377.624,Z 592.247,A -85,B 0,C 180,E1 -20169.61,E2 -20169.61} C_VEL
LIN {X 0,Y 379.967,Z 587.876,A -85,B 0,C 180,E1 -20171.699,E2 -20171.699} C_VEL
LIN {X 0,Y 382.064,Z 582.985,A -85,B 0,C 180,E1 -20173.427,E2 -20173.427} C_VEL
LIN {X 0,Y 384.628,Z 576.146,A -85,B 0,C 180,E1 -20175.311,E2 -20175.311} C_VEL
LIN {X 0,Y 387.36,Z 567.925,A -85,B 0,C 180,E1 -20177.088,E2 -20177.088} C_VEL
LIN {X 0,Y 389.855,Z 559.413,A -85,B 0,C 180,E1 -20178.597,E2 -20178.597} C_VEL
LIN {X 0,Y 392.647,Z 549.105,A -85,B 0,C 180,E1 -20180.084,E2 -20180.084} C_VEL
LIN {X 0,Y 395.379,Z 537.663,A -85,B 0,C 180,E1 -20181.431,E2 -20181.431} C_VEL
LIN {X 0,Y 397.671,Z 526.367,A -85,B 0,C 180,E1 -20182.525,E2 -20182.525} C_VEL
LIN {X 0,Y 399.988,Z 512.733,A -85,B 0,C 180,E1 -20183.614,E2 -20183.614} C_VEL
LIN {X 0,Y 401.899,Z 498.218,A -85,B 0,C 180,E1 -20184.518,E2 -20184.518} C_VEL
LIN {X 0,Y 403.265,Z 484.885,A -85,B 0,C 180,E1 -20185.162,E2 -20185.162} C_VEL
LIN {X 0,Y 405.004,Z 463.278,A -85,B 0,C 180,E1 -20185.929,E2 -20185.929} C_VEL
LIN {X 0,Y 411.084,Z 406.821,A -85,B 0,C 180,E1 -20187.692,E2 -20187.692} C_VEL
LIN {X 0,Y 406.057,Z 397.098,A -85,B 0,C 180,E1 -20189.255,E2 -20189.255} C_VEL
LIN {X 0,Y 401.963,Z 390.224,A -85,B 0,C 180,E1 -20190.645,E2 -20190.645} C_VEL
LIN {X 0,Y 399.534,Z 386.451,A -85,B 0,C 180,E1 -20191.535,E2 -20191.535} C_VEL
LIN {X 0,Y 397.208,Z 382.884,A -85,B 0,C 180,E1 -20192.467,E2 -20192.467} C_VEL
LIN {X 0,Y 394.728,Z 379.042,A -85,B 0,C 180,E1 -20193.603,E2 -20193.603} C_VEL
LIN {X 0,Y 392.281,Z 375.99,A -85,B 0,C 180,E1 -20194.778,E2 -20194.778} C_VEL
LIN {X 0,Y 391.476,Z 374.332,A -85,B 0,C 180,E1 -20195.285,E2 -20195.285} C_VEL
LIN {X 0,Y 388.868,Z 371.713,A -85,B 0,C 180,E1 -20196.832,E2 -20196.832} C_VEL
LIN {X 0,Y 387.44,Z 369.05,A -85,B 0,C 180,E1 -20198.102,E2 -20198.102} C_VEL
LIN {X 0,Y 384.677,Z 366.969,A -85,B 0,C 180,E1 -20201.303,E2 -20201.303} C_VEL
LIN {X 0,Y 384.174,Z 366.43,A -85,B 0,C 180,E1 -20203.172,E2 -20203.172} C_VEL
LIN {X 0,Y 384.584,Z 366.928,A -85,B 0,C 180,E1 -20205.446,E2 -20205.446} C_VEL
LIN {X 0,Y 386.44,Z 368.611,A -85,B 0,C 180,E1 -20208,E2 -20208} C_VEL
LIN {X 0,Y 387.381,Z 369.342,A -85,B 0,C 180,E1 -20208.864,E2 -20208.864} C_VEL
LIN {X 0,Y 388.896,Z 372.319,A -85,B 0,C 180,E1 -20210.194,E2 -20210.194} C_VEL
LIN {X 0,Y 391.276,Z 374.717,A -85,B 0,C 180,E1 -20211.636,E2 -20211.636} C_VEL
LIN {X 0,Y 392.689,Z 377.563,A -85,B 0,C 180,E1 -20212.513,E2 -20212.513} C_VEL
LIN {X 0,Y 395.581,Z 388.036,A -85,B 0,C 180,E1 -20214.451,E2 -20214.451} C_VEL
LIN {X 0,Y 399.651,Z 403.572,A -85,B 0,C 180,E1 -20216.717,E2 -20216.717} C_VEL
LIN {X 0,Y 400.54,Z 408.011,A -85,B 0,C 180,E1 -20217.221,E2 -20217.221} C_VEL
LIN {X 0,Y 402.071,Z 428.62,A -85,B 0,C 180,E1 -20218.794,E2 -20218.794} C_VEL
LIN {X 0,Y 403.419,Z 451.153,A -85,B 0,C 180,E1 -20220.292,E2 -20220.292} C_VEL
LIN {X 0,Y 403.963,Z 469.237,A -85,B 0,C 180,E1 -20221.305,E2 -20221.305} C_VEL
LIN {X 0,Y 403.669,Z 485.897,A -85,B 0,C 180,E1 -20222.063,E2 -20222.063} C_VEL
LIN {X 0,Y 397.934,Z 543.096,A -85,B 0,C 180,E1 -20223.858,E2 -20223.858} C_VEL
LIN {X 0,Y 395.609,Z 558.732,A -85,B 0,C 180,E1 -20224.503,E2 -20224.503} C_VEL
LIN {X 0,Y 393.112,Z 572.388,A -85,B 0,C 180,E1 -20225.246,E2 -20225.246} C_VEL
LIN {X 0,Y 390.18,Z 585.891,A -85,B 0,C 180,E1 -20226.177,E2 -20226.177} C_VEL
LIN {X 0,Y 386.799,Z 599.781,A -85,B 0,C 180,E1 -20227.368,E2 -20227.368} C_VEL
LIN {X 0,Y 383.907,Z 611.35,A -85,B 0,C 180,E1 -20228.598,E2 -20228.598} C_VEL
LIN {X 0,Y 380.883,Z 622.959,A -85,B 0,C 180,E1 -20230.11,E2 -20230.11} C_VEL
LIN {X 0,Y 377.896,Z 634.195,A -85,B 0,C 180,E1 -20231.912,E2 -20231.912} C_VEL
LIN {X 0,Y 375.747,Z 642.274,A -85,B 0,C 180,E1 -20233.484,E2 -20233.484} C_VEL
LIN {X 0,Y 373.88,Z 650.138,A -85,B 0,C 180,E1 -20235.35,E2 -20235.35} C_VEL
LIN {X 0,Y 372.511,Z 657.448,A -85,B 0,C 180,E1 -20237.512,E2 -20237.512} C_VEL
LIN {X 0,Y 371.955,Z 660.736,A -85,B 0,C 180,E1 -20238.642,E2 -20238.642} C_VEL
LIN {X 0,Y 371.525,Z 670.628,A -85,B 0,C 180,E1 -20240.231,E2 -20240.231} C_VEL
LIN {X 0,Y 371.087,Z 679.04,A -85,B 0,C 180,E1 -20241.861,E2 -20241.861} C_VEL
LIN {X 0,Y 370.946,Z 686.031,A -85,B 0,C 180,E1 -20243.494,E2 -20243.494} C_VEL
LIN {X 0,Y 370.806,Z 691.765,A -85,B 0,C 180,E1 -20245.124,E2 -20245.124} C_VEL
LIN {X 0,Y 370.697,Z 696.408,A -85,B 0,C 180,E1 -20246.75,E2 -20246.75} C_VEL
LIN {X 0,Y 370.662,Z 700.036,A -85,B 0,C 180,E1 -20248.376,E2 -20248.376} C_VEL
LIN {X 0,Y 370.681,Z 702.702,A -85,B 0,C 180,E1 -20250,E2 -20250} C_VEL
LIN {X 0,Y 370.62,Z 704.957,A -85,B 0,C 180,E1 -20252.166,E2 -20252.166} C_VEL
LIN {X 0,Y 370.713,Z 705.747,A -85,B 0,C 180,E1 -20254.334,E2 -20254.334} C_VEL
LIN {X 0,Y 371.168,Z 705.09,A -85,B 0,C 180,E1 -20256.501,E2 -20256.501} C_VEL
LIN {X 0,Y 371.927,Z 702.994,A -85,B 0,C 180,E1 -20258.665,E2 -20258.665} C_VEL
LIN {X 0,Y 373.142,Z 699.438,A -85,B 0,C 180,E1 -20260.819,E2 -20260.819} C_VEL
LIN {X 0,Y 375.114,Z 694.328,A -85,B 0,C 180,E1 -20262.948,E2 -20262.948} C_VEL
LIN {X 0,Y 377.151,Z 687.621,A -85,B 0,C 180,E1 -20265.07,E2 -20265.07} C_VEL
LIN {X 0,Y 379.585,Z 680.145,A -85,B 0,C 180,E1 -20266.896,E2 -20266.896} C_VEL
LIN {X 0,Y 382.437,Z 670.968,A -85,B 0,C 180,E1 -20268.694,E2 -20268.694} C_VEL
LIN {X 0,Y 385.142,Z 661.513,A -85,B 0,C 180,E1 -20270.215,E2 -20270.215} C_VEL
LIN {X 0,Y 388.226,Z 650.197,A -85,B 0,C 180,E1 -20271.707,E2 -20271.707} C_VEL
LIN {X 0,Y 391.389,Z 637.67,A -85,B 0,C 180,E1 -20273.047,E2 -20273.047} C_VEL
LIN {X 0,Y 394.157,Z 625.233,A -85,B 0,C 180,E1 -20274.125,E2 -20274.125} C_VEL
LIN {X 0,Y 397.192,Z 609.926,A -85,B 0,C 180,E1 -20275.179,E2 -20275.179} C_VEL
LIN {X 0,Y 399.815,Z 594.316,A -85,B 0,C 180,E1 -20275.975,E2 -20275.975} C_VEL
LIN {X 0,Y 402.005,Z 577.78,A -85,B 0,C 180,E1 -20276.588,E2 -20276.588} C_VEL
LIN {X 0,Y 411.827,Z 491.062,A -85,B 0,C 180,E1 -20279.34,E2 -20279.34} C_VEL
LIN {X 0,Y 412.433,Z 484.321,A -85,B 0,C 180,E1 -20279.599,E2 -20279.599} C_VEL
LIN {X 0,Y 412.64,Z 468.348,A -85,B 0,C 180,E1 -20280.466,E2 -20280.466} C_VEL
LIN {X 0,Y 412.378,Z 454.106,A -85,B 0,C 180,E1 -20281.383,E2 -20281.383} C_VEL
LIN {X 0,Y 411.644,Z 438.076,A -85,B 0,C 180,E1 -20282.606,E2 -20282.606} C_VEL
LIN {X 0,Y 413.843,Z 425.137,A -85,B 0,C 180,E1 -20284.094,E2 -20284.094} C_VEL
LIN {X 0,Y 414.846,Z 420.057,A -85,B 0,C 180,E1 -20284.727,E2 -20284.727} C_VEL
LIN {X 0,Y 414.694,Z 418.667,A -85,B 0,C 180,E1 -20285.049,E2 -20285.049} C_VEL
LIN {X 0,Y 412.229,Z 414.546,A -85,B 0,C 180,E1 -20287.003,E2 -20287.003} C_VEL
LIN {X 0,Y 410.126,Z 411.575,A -85,B 0,C 180,E1 -20289.191,E2 -20289.191} C_VEL
LIN {X 0,Y 408.782,Z 410.283,A -85,B 0,C 180,E1 -20291.068,E2 -20291.068} C_VEL
LIN {X 0,Y 407.877,Z 409.908,A -85,B 0,C 180,E1 -20293.387,E2 -20293.387} C_VEL
LIN {X 0,Y 407.653,Z 410.66,A -85,B 0,C 180,E1 -20295.213,E2 -20295.213} C_VEL
LIN {X 0,Y 407.646,Z 411.888,A -85,B 0,C 180,E1 -20296.583,E2 -20296.583} C_VEL
LIN {X 0,Y 408.066,Z 415.426,A -85,B 0,C 180,E1 -20299.048,E2 -20299.048} C_VEL
LIN {X 0,Y 408.696,Z 420.07,A -85,B 0,C 180,E1 -20301.248,E2 -20301.248} C_VEL
LIN {X 0,Y 409.286,Z 425.499,A -85,B 0,C 180,E1 -20303.203,E2 -20303.203} C_VEL
LIN {X 0,Y 409.635,Z 432.336,A -85,B 0,C 180,E1 -20305.161,E2 -20305.161} C_VEL
LIN {X 0,Y 409.637,Z 433.336,A -85,B 0,C 180,E1 -20305.411,E2 -20305.411} C_VEL
LIN {X 0,Y 407.852,Z 440.075,A -85,B 0,C 180,E1 -20306.472,E2 -20306.472} C_VEL
LIN {X 0,Y 409.517,Z 455.422,A -85,B 0,C 180,E1 -20307.959,E2 -20307.959} C_VEL
LIN {X 0,Y 410.876,Z 469.28,A -85,B 0,C 180,E1 -20309.134,E2 -20309.134} C_VEL
LIN {X 0,Y 411.953,Z 482.718,A -85,B 0,C 180,E1 -20310.13,E2 -20310.13} C_VEL
LIN {X 0,Y 412.248,Z 490.287,A -85,B 0,C 180,E1 -20310.599,E2 -20310.599} C_VEL
LIN {X 0,Y 401.477,Z 584.759,A -85,B 0,C 180,E1 -20313.584,E2 -20313.584} C_VEL
LIN {X 0,Y 398.959,Z 601.059,A -85,B 0,C 180,E1 -20314.315,E2 -20314.315} C_VEL
LIN {X 0,Y 396.36,Z 615.402,A -85,B 0,C 180,E1 -20315.184,E2 -20315.184} C_VEL
LIN {X 0,Y 393.463,Z 629.153,A -85,B 0,C 180,E1 -20316.249,E2 -20316.249} C_VEL
LIN {X 0,Y 390.506,Z 641.722,A -85,B 0,C 180,E1 -20317.456,E2 -20317.456} C_VEL
LIN {X 0,Y 387.442,Z 653.295,A -85,B 0,C 180,E1 -20318.803,E2 -20318.803} C_VEL
LIN {X 0,Y 384.461,Z 663.76,A -85,B 0,C 180,E1 -20320.303,E2 -20320.303} C_VEL
LIN {X 0,Y 381.403,Z 673.913,A -85,B 0,C 180,E1 -20322.085,E2 -20322.085} C_VEL
LIN {X 0,Y 378.753,Z 682.232,A -85,B 0,C 180,E1 -20323.895,E2 -20323.895} C_VEL
LIN {X 0,Y 376.8,Z 688.091,A -85,B 0,C 180,E1 -20325.466,E2 -20325.466} C_VEL
LIN {X 0,Y 375.312,Z 692.927,A -85,B 0,C 180,E1 -20327.059,E2 -20327.059} C_VEL
LIN {X 0,Y 373.795,Z 696.902,A -85,B 0,C 180,E1 -20328.653,E2 -20328.653} C_VEL
LIN {X 0,Y 372.633,Z 699.933,A -85,B 0,C 180,E1 -20330.26,E2 -20330.26} C_VEL
LIN {X 0,Y 371.595,Z 702.726,A -85,B 0,C 180,E1 -20332.418,E2 -20332.418} C_VEL
LIN {X 0,Y 370.921,Z 704.096,A -85,B 0,C 180,E1 -20334.582,E2 -20334.582} C_VEL
LIN {X 0,Y 370.582,Z 704.027,A -85,B 0,C 180,E1 -20336.75,E2 -20336.75} C_VEL
LIN {X 0,Y 370.527,Z 702.519,A -85,B 0,C 180,E1 -20338.917,E2 -20338.917} C_VEL
LIN {X 0,Y 370.582,Z 701.219,A -85,B 0,C 180,E1 -20340,E2 -20340} C_VEL
LIN {X 0,Y 370.626,Z 697.474,A -85,B 0,C 180,E1 -20342.166,E2 -20342.166} C_VEL
LIN {X 0,Y 370.659,Z 693.581,A -85,B 0,C 180,E1 -20343.793,E2 -20343.793} C_VEL
LIN {X 0,Y 370.785,Z 688.685,A -85,B 0,C 180,E1 -20345.42,E2 -20345.42} C_VEL
LIN {X 0,Y 371.042,Z 681.52,A -85,B 0,C 180,E1 -20347.321,E2 -20347.321} C_VEL
LIN {X 0,Y 371.455,Z 672.607,A -85,B 0,C 180,E1 -20349.224,E2 -20349.224} C_VEL
LIN {X 0,Y 371.953,Z 663.284,A -85,B 0,C 180,E1 -20350.855,E2 -20350.855} C_VEL
LIN {X 0,Y 372.605,Z 653.477,A -85,B 0,C 180,E1 -20352.285,E2 -20352.285} C_VEL
LIN {X 0,Y 373.291,Z 641.766,A -85,B 0,C 180,E1 -20353.704,E2 -20353.704} C_VEL
LIN {X 0,Y 374.169,Z 628.079,A -85,B 0,C 180,E1 -20355.055,E2 -20355.055} C_VEL
LIN {X 0,Y 375.041,Z 614.562,A -85,B 0,C 180,E1 -20356.13,E2 -20356.13} C_VEL
LIN {X 0,Y 375.671,Z 600.449,A -85,B 0,C 180,E1 -20357.008,E2 -20357.008} C_VEL
LIN {X 0,Y 376.426,Z 584.63,A -85,B 0,C 180,E1 -20357.741,E2 -20357.741} C_VEL
LIN {X 0,Y 377.044,Z 565.417,A -85,B 0,C 180,E1 -20358.34,E2 -20358.34} C_VEL
LIN {X 0,Y 379.802,Z 474.216,A -85,B 0,C 180,E1 -20360.901,E2 -20360.901} C_VEL
LIN {X 0,Y 377.19,Z 443.852,A -85,B 0,C 180,E1 -20361.845,E2 -20361.845} C_VEL
LIN {X 0,Y 377.046,Z 439.445,A -85,B 0,C 180,E1 -20362.005,E2 -20362.005} C_VEL
LIN {X 0,Y 379.139,Z 411.343,A -85,B 0,C 180,E1 -20365.879,E2 -20365.879} C_VEL
LIN {X 0,Y 381.029,Z 387.608,A -85,B 0,C 180,E1 -20369.154,E2 -20369.154} C_VEL
LIN {X 0,Y 377.316,Z 370.208,A -85,B 0,C 180,E1 -20371.794,E2 -20371.794} C_VEL
LIN {X 0,Y 373.112,Z 351.568,A -85,B 0,C 180,E1 -20374.725,E2 -20374.725} C_VEL
LIN {X 0,Y 373.046,Z 351.572,A -85,B 0,C 180,E1 -20378.289,E2 -20378.289} C_VEL
LIN {X 0,Y 373.016,Z 351.577,A -85,B 0,C 180,E1 -20381.313,E2 -20381.313} C_VEL
LIN {X 0,Y 373.09,Z 351.567,A -85,B 0,C 180,E1 -20384.486,E2 -20384.486} C_VEL
LIN {X 0,Y 373.043,Z 351.573,A -85,B 0,C 180,E1 -20387.472,E2 -20387.472} C_VEL
LIN {X 0,Y 373.039,Z 351.57,A -85,B 0,C 180,E1 -20390.341,E2 -20390.341} C_VEL
LIN {X 0,Y 373.069,Z 351.565,A -85,B 0,C 180,E1 -20393.837,E2 -20393.837} C_VEL
LIN {X 0,Y 373.023,Z 351.57,A -85,B 0,C 180,E1 -20397.006,E2 -20397.006} C_VEL
LIN {X 0,Y 373.077,Z 351.565,A -85,B 0,C 180,E1 -20399.729,E2 -20399.729} C_VEL
LIN {X 0,Y 373.087,Z 351.568,A -85,B 0,C 180,E1 -20403.219,E2 -20403.219} C_VEL
LIN {X 0,Y 373.09,Z 351.568,A -85,B 0,C 180,E1 -20406.917,E2 -20406.917} C_VEL
LIN {X 0,Y 373.126,Z 351.569,A -85,B 0,C 180,E1 -20410.599,E2 -20410.599} C_VEL
LIN {X 0,Y 374.196,Z 354.483,A -85,B 0,C 180,E1 -20410.738,E2 -20410.738} C_VEL
LIN {X 0,Y 384.693,Z 379.541,A -85,B 0,C 180,E1 -20411.893,E2 -20411.893} C_VEL
LIN {X 0,Y 385.495,Z 381.675,A -85,B 0,C 180,E1 -20411.982,E2 -20411.982} C_VEL
LIN {X 0,Y 384.081,Z 456.894,A -85,B 0,C 180,E1 -20413.376,E2 -20413.376} C_VEL
LIN {X 0,Y 383.929,Z 474.33,A -85,B 0,C 180,E1 -20413.778,E2 -20413.778} C_VEL
LIN {X 0,Y 383.475,Z 488.251,A -85,B 0,C 180,E1 -20414.302,E2 -20414.302} C_VEL
LIN {X 0,Y 382.783,Z 501.741,A -85,B 0,C 180,E1 -20415.021,E2 -20415.021} C_VEL
LIN {X 0,Y 381.785,Z 514.785,A -85,B 0,C 180,E1 -20415.931,E2 -20415.931} C_VEL
LIN {X 0,Y 380.824,Z 526.574,A -85,B 0,C 180,E1 -20416.979,E2 -20416.979} C_VEL
LIN {X 0,Y 379.614,Z 538.516,A -85,B 0,C 180,E1 -20418.29,E2 -20418.29} C_VEL
LIN {X 0,Y 378.312,Z 548.423,A -85,B 0,C 180,E1 -20419.6,E2 -20419.6} C_VEL
LIN {X 0,Y 376.969,Z 558.268,A -85,B 0,C 180,E1 -20421.182,E2 -20421.182} C_VEL
LIN {X 0,Y 375.828,Z 566.445,A -85,B 0,C 180,E1 -20422.773,E2 -20422.773} C_VEL
LIN {X 0,Y 374.703,Z 574.268,A -85,B 0,C 180,E1 -20424.637,E2 -20424.637} C_VEL
LIN {X 0,Y 373.878,Z 579.789,A -85,B 0,C 180,E1 -20426.241,E2 -20426.241} C_VEL
LIN {X 0,Y 373.156,Z 585.562,A -85,B 0,C 180,E1 -20428.387,E2 -20428.387} C_VEL
LIN {X 0,Y 372.753,Z 588.915,A -85,B 0,C 180,E1 -20430,E2 -20430} C_VEL
LIN {X 0,Y 372.483,Z 592.099,A -85,B 0,C 180,E1 -20432.156,E2 -20432.156} C_VEL
LIN {X 0,Y 372.383,Z 593.945,A -85,B 0,C 180,E1 -20434.315,E2 -20434.315} C_VEL
LIN {X 0,Y 372.546,Z 594.495,A -85,B 0,C 180,E1 -20436.477,E2 -20436.477} C_VEL
LIN {X 0,Y 372.915,Z 593.756,A -85,B 0,C 180,E1 -20438.642,E2 -20438.642} C_VEL
LIN {X 0,Y 373.435,Z 591.716,A -85,B 0,C 180,E1 -20440.811,E2 -20440.811} C_VEL
LIN {X 0,Y 374.485,Z 588.273,A -85,B 0,C 180,E1 -20442.971,E2 -20442.971} C_VEL
LIN {X 0,Y 375.693,Z 583.356,A -85,B 0,C 180,E1 -20445.131,E2 -20445.131} C_VEL
LIN {X 0,Y 376.838,Z 578.566,A -85,B 0,C 180,E1 -20446.745,E2 -20446.745} C_VEL
LIN {X 0,Y 378.399,Z 571.651,A -85,B 0,C 180,E1 -20448.621,E2 -20448.621} C_VEL
LIN {X 0,Y 380.212,Z 563.05,A -85,B 0,C 180,E1 -20450.489,E2 -20450.489} C_VEL
LIN {X 0,Y 382.008,Z 554.01,A -85,B 0,C 180,E1 -20452.079,E2 -20452.079} C_VEL
LIN {X 0,Y 383.61,Z 544.961,A -85,B 0,C 180,E1 -20453.4,E2 -20453.4} C_VEL
LIN {X 0,Y 385.236,Z 534.128,A -85,B 0,C 180,E1 -20454.721,E2 -20454.721} C_VEL
LIN {X 0,Y 386.951,Z 522.204,A -85,B 0,C 180,E1 -20455.894,E2 -20455.894} C_VEL
LIN {X 0,Y 388.248,Z 510.704,A -85,B 0,C 180,E1 -20456.81,E2 -20456.81} C_VEL
LIN {X 0,Y 389.08,Z 499.412,A -85,B 0,C 180,E1 -20457.545,E2 -20457.545} C_VEL
LIN {X 0,Y 389.933,Z 485.721,A -85,B 0,C 180,E1 -20458.221,E2 -20458.221} C_VEL
LIN {X 0,Y 390.414,Z 470.993,A -85,B 0,C 180,E1 -20458.725,E2 -20458.725} C_VEL
LIN {X 0,Y 391.652,Z 418.212,A -85,B 0,C 180,E1 -20459.725,E2 -20459.725} C_VEL
LIN {X 0,Y 392.242,Z 390.756,A -85,B 0,C 180,E1 -20460.237,E2 -20460.237} C_VEL
LIN {X 0,Y 382.487,Z 370.132,A -85,B 0,C 180,E1 -20461.454,E2 -20461.454} C_VEL
LIN {X 0,Y 374.624,Z 355.277,A -85,B 0,C 180,E1 -20462.454,E2 -20462.454} C_VEL
LIN {X 0,Y 372.358,Z 353.487,A -85,B 0,C 180,E1 -20462.812,E2 -20462.812} C_VEL
LIN {X 0,Y 370.434,Z 352.569,A -85,B 0,C 180,E1 -20463.291,E2 -20463.291} C_VEL
LIN {X 0,Y 368.261,Z 352.212,A -85,B 0,C 180,E1 -20464.136,E2 -20464.136} C_VEL
LIN {X 0,Y 366.349,Z 352.408,A -85,B 0,C 180,E1 -20465.75,E2 -20465.75} C_VEL
LIN {X 0,Y 365.947,Z 352.456,A -85,B 0,C 180,E1 -20467.091,E2 -20467.091} C_VEL
LIN {X 0,Y 365.93,Z 352.465,A -85,B 0,C 180,E1 -20470.603,E2 -20470.603} C_VEL
LIN {X 0,Y 365.959,Z 352.461,A -85,B 0,C 180,E1 -20473.555,E2 -20473.555} C_VEL
LIN {X 0,Y 365.969,Z 352.457,A -85,B 0,C 180,E1 -20476.661,E2 -20476.661} C_VEL
LIN {X 0,Y 365.957,Z 352.457,A -85,B 0,C 180,E1 -20479.961,E2 -20479.961} C_VEL
LIN {X 0,Y 365.992,Z 352.41,A -85,B 0,C 180,E1 -20483.609,E2 -20483.609} C_VEL
LIN {X 0,Y 365.936,Z 352.453,A -85,B 0,C 180,E1 -20486.282,E2 -20486.282} C_VEL
LIN {X 0,Y 365.975,Z 352.442,A -85,B 0,C 180,E1 -20489.459,E2 -20489.459} C_VEL
LIN {X 0,Y 366.014,Z 352.445,A -85,B 0,C 180,E1 -20492.658,E2 -20492.658} C_VEL
LIN {X 0,Y 366,Z 352.443,A -85,B 0,C 180,E1 -20495.1,E2 -20495.1} C_VEL
LIN {X 0,Y 366.057,Z 352.438,A -85,B 0,C 180,E1 -20497.886,E2 -20497.886} C_VEL
LIN {X 0,Y 372.158,Z 374.801,A -85,B 0,C 180,E1 -20498.706,E2 -20498.706} C_VEL
LIN {X 0,Y 369.821,Z 469.591,A -85,B 0,C 180,E1 -20501.409,E2 -20501.409} C_VEL
LIN {X 0,Y 369.505,Z 484.835,A -85,B 0,C 180,E1 -20502.059,E2 -20502.059} C_VEL
LIN {X 0,Y 368.955,Z 499.27,A -85,B 0,C 180,E1 -20502.886,E2 -20502.886} C_VEL
LIN {X 0,Y 368.277,Z 514.065,A -85,B 0,C 180,E1 -20503.991,E2 -20503.991} C_VEL
LIN {X 0,Y 367.585,Z 527.429,A -85,B 0,C 180,E1 -20505.234,E2 -20505.234} C_VEL
LIN {X 0,Y 366.947,Z 539.569,A -85,B 0,C 180,E1 -20506.617,E2 -20506.617} C_VEL
LIN {X 0,Y 366.346,Z 550.625,A -85,B 0,C 180,E1 -20508.139,E2 -20508.139} C_VEL
LIN {X 0,Y 365.771,Z 560.689,A -85,B 0,C 180,E1 -20509.797,E2 -20509.797} C_VEL
LIN {X 0,Y 365.357,Z 569.103,A -85,B 0,C 180,E1 -20511.455,E2 -20511.455} C_VEL
LIN {X 0,Y 365.033,Z 577.208,A -85,B 0,C 180,E1 -20513.388,E2 -20513.388} C_VEL
LIN {X 0,Y 364.958,Z 582.859,A -85,B 0,C 180,E1 -20515.045,E2 -20515.045} C_VEL
LIN {X 0,Y 365.016,Z 587.469,A -85,B 0,C 180,E1 -20516.699,E2 -20516.699} C_VEL
LIN {X 0,Y 365.169,Z 592.216,A -85,B 0,C 180,E1 -20518.901,E2 -20518.901} C_VEL
LIN {X 0,Y 365.644,Z 595.386,A -85,B 0,C 180,E1 -20521.097,E2 -20521.097} C_VEL
LIN {X 0,Y 366.405,Z 597.123,A -85,B 0,C 180,E1 -20523.287,E2 -20523.287} C_VEL
LIN {X 0,Y 367.517,Z 597.44,A -85,B 0,C 180,E1 -20525.468,E2 -20525.468} C_VEL
LIN {X 0,Y 368.909,Z 596.359,A -85,B 0,C 180,E1 -20527.637,E2 -20527.637} C_VEL
LIN {X 0,Y 370.788,Z 593.784,A -85,B 0,C 180,E1 -20529.789,E2 -20529.789} C_VEL
LIN {X 0,Y 373.23,Z 589.637,A -85,B 0,C 180,E1 -20531.913,E2 -20531.913} C_VEL
LIN {X 0,Y 375.891,Z 583.93,A -85,B 0,C 180,E1 -20534.019,E2 -20534.019} C_VEL
LIN {X 0,Y 378.463,Z 577.556,A -85,B 0,C 180,E1 -20535.808,E2 -20535.808} C_VEL
LIN {X 0,Y 381.391,Z 569.315,A -85,B 0,C 180,E1 -20537.64,E2 -20537.64} C_VEL
LIN {X 0,Y 384.504,Z 559.348,A -85,B 0,C 180,E1 -20539.418,E2 -20539.418} C_VEL
LIN {X 0,Y 387.492,Z 548.819,A -85,B 0,C 180,E1 -20540.916,E2 -20540.916} C_VEL
LIN {X 0,Y 390.37,Z 537.158,A -85,B 0,C 180,E1 -20542.275,E2 -20542.275} C_VEL
LIN {X 0,Y 393.154,Z 524.196,A -85,B 0,C 180,E1 -20543.493,E2 -20543.493} C_VEL
LIN {X 0,Y 395.285,Z 511.574,A -85,B 0,C 180,E1 -20544.469,E2 -20544.469} C_VEL
LIN {X 0,Y 397.225,Z 497.276,A -85,B 0,C 180,E1 -20545.345,E2 -20545.345} C_VEL
LIN {X 0,Y 398.718,Z 482.8,A -85,B 0,C 180,E1 -20546.019,E2 -20546.019} C_VEL
LIN {X 0,Y 400.626,Z 461.644,A -85,B 0,C 180,E1 -20546.757,E2 -20546.757} C_VEL
LIN {X 0,Y 406.514,Z 410.229,A -85,B 0,C 180,E1 -20548.396,E2 -20548.396} C_VEL
LIN {X 0,Y 401.664,Z 400.777,A -85,B 0,C 180,E1 -20550.016,E2 -20550.016} C_VEL
LIN {X 0,Y 397.285,Z 393.311,A -85,B 0,C 180,E1 -20551.659,E2 -20551.659} C_VEL
LIN {X 0,Y 394.492,Z 389,A -85,B 0,C 180,E1 -20552.816,E2 -20552.816} C_VEL
LIN {X 0,Y 391.983,Z 385.171,A -85,B 0,C 180,E1 -20554.003,E2 -20554.003} C_VEL
LIN {X 0,Y 389.724,Z 381.974,A -85,B 0,C 180,E1 -20555.205,E2 -20555.205} C_VEL
LIN {X 0,Y 389.025,Z 380.786,A -85,B 0,C 180,E1 -20555.641,E2 -20555.641} C_VEL
LIN {X 0,Y 386.499,Z 377.773,A -85,B 0,C 180,E1 -20557.322,E2 -20557.322} C_VEL
LIN {X 0,Y 385.52,Z 375.801,A -85,B 0,C 180,E1 -20558.256,E2 -20558.256} C_VEL
LIN {X 0,Y 382.918,Z 373.818,A -85,B 0,C 180,E1 -20561.411,E2 -20561.411} C_VEL
LIN {X 0,Y 382.466,Z 373.342,A -85,B 0,C 180,E1 -20562.898,E2 -20562.898} C_VEL
LIN {X 0,Y 382.825,Z 373.769,A -85,B 0,C 180,E1 -20565.356,E2 -20565.356} C_VEL
LIN {X 0,Y 384.658,Z 375.475,A -85,B 0,C 180,E1 -20567.954,E2 -20567.954} C_VEL
LIN {X 0,Y 385.406,Z 376.126,A -85,B 0,C 180,E1 -20568.673,E2 -20568.673} C_VEL
LIN {X 0,Y 386.958,Z 379.1,A -85,B 0,C 180,E1 -20570.077,E2 -20570.077} C_VEL
LIN {X 0,Y 388.954,Z 381.203,A -85,B 0,C 180,E1 -20571.358,E2 -20571.358} C_VEL
LIN {X 0,Y 390.161,Z 383.855,A -85,B 0,C 180,E1 -20572.15,E2 -20572.15} C_VEL
LIN {X 0,Y 392.506,Z 393.201,A -85,B 0,C 180,E1 -20573.898,E2 -20573.898} C_VEL
LIN {X 0,Y 396.172,Z 408.343,A -85,B 0,C 180,E1 -20576.147,E2 -20576.147} C_VEL
LIN {X 0,Y 396.761,Z 411.699,A -85,B 0,C 180,E1 -20576.536,E2 -20576.536} C_VEL
LIN {X 0,Y 397.95,Z 432.426,A -85,B 0,C 180,E1 -20578.149,E2 -20578.149} C_VEL
LIN {X 0,Y 398.963,Z 453.63,A -85,B 0,C 180,E1 -20579.587,E2 -20579.587} C_VEL
LIN {X 0,Y 399.291,Z 470.87,A -85,B 0,C 180,E1 -20580.581,E2 -20580.581} C_VEL
LIN {X 0,Y 398.925,Z 486.559,A -85,B 0,C 180,E1 -20581.318,E2 -20581.318} C_VEL
LIN {X 0,Y 392.955,Z 542.484,A -85,B 0,C 180,E1 -20583.108,E2 -20583.108} C_VEL
LIN {X 0,Y 390.439,Z 558.284,A -85,B 0,C 180,E1 -20583.782,E2 -20583.782} C_VEL
LIN {X 0,Y 387.623,Z 572.486,A -85,B 0,C 180,E1 -20584.585,E2 -20584.585} C_VEL
LIN {X 0,Y 384.209,Z 587.31,A -85,B 0,C 180,E1 -20585.639,E2 -20585.639} C_VEL
LIN {X 0,Y 380.728,Z 600.723,A -85,B 0,C 180,E1 -20586.843,E2 -20586.843} C_VEL
LIN {X 0,Y 377.438,Z 612.835,A -85,B 0,C 180,E1 -20588.213,E2 -20588.213} C_VEL
LIN {X 0,Y 374.776,Z 622.318,A -85,B 0,C 180,E1 -20589.486,E2 -20589.486} C_VEL
LIN {X 0,Y 372.022,Z 631.991,A -85,B 0,C 180,E1 -20591.047,E2 -20591.047} C_VEL
LIN {X 0,Y 369.261,Z 641.438,A -85,B 0,C 180,E1 -20592.901,E2 -20592.901} C_VEL
LIN {X 0,Y 367.258,Z 649.277,A -85,B 0,C 180,E1 -20594.797,E2 -20594.797} C_VEL
LIN {X 0,Y 365.851,Z 655.67,A -85,B 0,C 180,E1 -20596.718,E2 -20596.718} C_VEL
LIN {X 0,Y 364.848,Z 661.323,A -85,B 0,C 180,E1 -20598.795,E2 -20598.795} C_VEL
LIN {X 0,Y 364.42,Z 670.583,A -85,B 0,C 180,E1 -20600.318,E2 -20600.318} C_VEL
LIN {X 0,Y 363.988,Z 679.011,A -85,B 0,C 180,E1 -20601.98,E2 -20601.98} C_VEL
LIN {X 0,Y 363.85,Z 686.005,A -85,B 0,C 180,E1 -20603.645,E2 -20603.645} C_VEL
LIN {X 0,Y 363.715,Z 692.578,A -85,B 0,C 180,E1 -20605.582,E2 -20605.582} C_VEL
LIN {X 0,Y 363.63,Z 697.018,A -85,B 0,C 180,E1 -20607.24,E2 -20607.24} C_VEL
LIN {X 0,Y 363.608,Z 700.499,A -85,B 0,C 180,E1 -20608.896,E2 -20608.896} C_VEL
LIN {X 0,Y 363.597,Z 702.285,A -85,B 0,C 180,E1 -20610,E2 -20610} C_VEL
LIN {X 0,Y 363.524,Z 704.709,A -85,B 0,C 180,E1 -20612.208,E2 -20612.208} C_VEL
LIN {X 0,Y 363.635,Z 705.683,A -85,B 0,C 180,E1 -20614.419,E2 -20614.419} C_VEL
LIN {X 0,Y 364.1,Z 705.227,A -85,B 0,C 180,E1 -20616.628,E2 -20616.628} C_VEL
LIN {X 0,Y 364.902,Z 703.36,A -85,B 0,C 180,E1 -20618.833,E2 -20618.833} C_VEL
LIN {X 0,Y 366.212,Z 700.056,A -85,B 0,C 180,E1 -20621.027,E2 -20621.027} C_VEL
LIN {X 0,Y 368.254,Z 695.175,A -85,B 0,C 180,E1 -20623.194,E2 -20623.194} C_VEL
LIN {X 0,Y 370.393,Z 688.707,A -85,B 0,C 180,E1 -20625.352,E2 -20625.352} C_VEL
LIN {X 0,Y 372.92,Z 681.542,A -85,B 0,C 180,E1 -20627.207,E2 -20627.207} C_VEL
LIN {X 0,Y 375.919,Z 672.749,A -85,B 0,C 180,E1 -20629.031,E2 -20629.031} C_VEL
LIN {X 0,Y 378.732,Z 663.677,A -85,B 0,C 180,E1 -20630.573,E2 -20630.573} C_VEL
LIN {X 0,Y 381.917,Z 652.837,A -85,B 0,C 180,E1 -20632.084,E2 -20632.084} C_VEL
LIN {X 0,Y 385.179,Z 640.871,A -85,B 0,C 180,E1 -20633.44,E2 -20633.44} C_VEL
LIN {X 0,Y 388.357,Z 627.827,A -85,B 0,C 180,E1 -20634.651,E2 -20634.651} C_VEL
LIN {X 0,Y 391.172,Z 615.033,A -85,B 0,C 180,E1 -20635.594,E2 -20635.594} C_VEL
LIN {X 0,Y 393.628,Z 602.261,A -85,B 0,C 180,E1 -20636.343,E2 -20636.343} C_VEL
LIN {X 0,Y 396.04,Z 587.113,A -85,B 0,C 180,E1 -20637.021,E2 -20637.021} C_VEL
LIN {X 0,Y 408.023,Z 488.35,A -85,B 0,C 180,E1 -20640.244,E2 -20640.244} C_VEL
LIN {X 0,Y 408.443,Z 476.977,A -85,B 0,C 180,E1 -20640.836,E2 -20640.836} C_VEL
LIN {X 0,Y 408.547,Z 461.487,A -85,B 0,C 180,E1 -20641.79,E2 -20641.79} C_VEL
LIN {X 0,Y 408.065,Z 442.885,A -85,B 0,C 180,E1 -20643.189,E2 -20643.189} C_VEL
LIN {X 0,Y 407.855,Z 438.072,A -85,B 0,C 180,E1 -20643.613,E2 -20643.613} C_VEL
LIN {X 0,Y 410.504,Z 425.274,A -85,B 0,C 180,E1 -20645.136,E2 -20645.136} C_VEL
LIN {X 0,Y 410.445,Z 423.838,A -85,B 0,C 180,E1 -20645.466,E2 -20645.466} C_VEL
LIN {X 0,Y 408.688,Z 420.904,A -85,B 0,C 180,E1 -20646.86,E2 -20646.86} C_VEL
LIN {X 0,Y 407.173,Z 418.688,A -85,B 0,C 180,E1 -20648.265,E2 -20648.265} C_VEL
LIN {X 0,Y 405.332,Z 416.562,A -85,B 0,C 180,E1 -20650.505,E2 -20650.505} C_VEL
LIN {X 0,Y 404.28,Z 415.855,A -85,B 0,C 180,E1 -20652.509,E2 -20652.509} C_VEL
LIN {X 0,Y 403.749,Z 416.229,A -85,B 0,C 180,E1 -20654.66,E2 -20654.66} C_VEL
LIN {X 0,Y 403.564,Z 418.016,A -85,B 0,C 180,E1 -20656.8,E2 -20656.8} C_VEL
LIN {X 0,Y 403.744,Z 420.744,A -85,B 0,C 180,E1 -20658.757,E2 -20658.757} C_VEL
LIN {X 0,Y 404.115,Z 424.643,A -85,B 0,C 180,E1 -20660.725,E2 -20660.725} C_VEL
LIN {X 0,Y 404.566,Z 430.045,A -85,B 0,C 180,E1 -20662.79,E2 -20662.79} C_VEL
LIN {X 0,Y 404.75,Z 437.044,A -85,B 0,C 180,E1 -20664.865,E2 -20664.865} C_VEL
LIN {X 0,Y 404.109,Z 440.091,A -85,B 0,C 180,E1 -20665.37,E2 -20665.37} C_VEL
LIN {X 0,Y 405.533,Z 456.153,A -85,B 0,C 180,E1 -20667.009,E2 -20667.009} C_VEL
LIN {X 0,Y 406.801,Z 471.191,A -85,B 0,C 180,E1 -20668.345,E2 -20668.345} C_VEL
LIN {X 0,Y 407.74,Z 485.544,A -85,B 0,C 180,E1 -20669.438,E2 -20669.438} C_VEL
LIN {X 0,Y 407.877,Z 491.944,A -85,B 0,C 180,E1 -20669.841,E2 -20669.841} C_VEL
LIN {X 0,Y 396.626,Z 585.109,A -85,B 0,C 180,E1 -20672.845,E2 -20672.845} C_VEL
LIN {X 0,Y 394.079,Z 600.677,A -85,B 0,C 180,E1 -20673.547,E2 -20673.547} C_VEL
LIN {X 0,Y 391.365,Z 614.997,A -85,B 0,C 180,E1 -20674.42,E2 -20674.42} C_VEL
LIN {X 0,Y 388.248,Z 628.787,A -85,B 0,C 180,E1 -20675.484,E2 -20675.484} C_VEL
LIN {X 0,Y 385.129,Z 641.336,A -85,B 0,C 180,E1 -20676.698,E2 -20676.698} C_VEL
LIN {X 0,Y 382.187,Z 651.938,A -85,B 0,C 180,E1 -20677.932,E2 -20677.932} C_VEL
LIN {X 0,Y 379.016,Z 662.63,A -85,B 0,C 180,E1 -20679.444,E2 -20679.444} C_VEL
LIN {X 0,Y 376.12,Z 671.625,A -85,B 0,C 180,E1 -20680.98,E2 -20680.98} C_VEL
LIN {X 0,Y 373.198,Z 680.301,A -85,B 0,C 180,E1 -20682.806,E2 -20682.806} C_VEL
LIN {X 0,Y 370.688,Z 687.394,A -85,B 0,C 180,E1 -20684.661,E2 -20684.661} C_VEL
LIN {X 0,Y 368.468,Z 693.804,A -85,B 0,C 180,E1 -20686.814,E2 -20686.814} C_VEL
LIN {X 0,Y 366.379,Z 698.645,A -85,B 0,C 180,E1 -20688.979,E2 -20688.979} C_VEL
LIN {X 0,Y 365.058,Z 701.926,A -85,B 0,C 180,E1 -20691.171,E2 -20691.171} C_VEL
LIN {X 0,Y 364.149,Z 703.771,A -85,B 0,C 180,E1 -20693.373,E2 -20693.373} C_VEL
LIN {X 0,Y 363.633,Z 704.216,A -85,B 0,C 180,E1 -20695.581,E2 -20695.581} C_VEL
LIN {X 0,Y 363.454,Z 703.244,A -85,B 0,C 180,E1 -20697.791,E2 -20697.791} C_VEL
LIN {X 0,Y 363.5,Z 700.836,A -85,B 0,C 180,E1 -20700,E2 -20700} C_VEL
LIN {X 0,Y 363.565,Z 696.907,A -85,B 0,C 180,E1 -20702.209,E2 -20702.209} C_VEL
LIN {X 0,Y 363.603,Z 692.824,A -85,B 0,C 180,E1 -20703.866,E2 -20703.866} C_VEL
LIN {X 0,Y 363.734,Z 687.737,A -85,B 0,C 180,E1 -20705.526,E2 -20705.526} C_VEL
LIN {X 0,Y 363.967,Z 680.359,A -85,B 0,C 180,E1 -20707.464,E2 -20707.464} C_VEL
LIN {X 0,Y 364.336,Z 672.591,A -85,B 0,C 180,E1 -20709.126,E2 -20709.126} C_VEL
LIN {X 0,Y 364.84,Z 663.252,A -85,B 0,C 180,E1 -20710.789,E2 -20710.789} C_VEL
LIN {X 0,Y 365.584,Z 652.348,A -85,B 0,C 180,E1 -20712.394,E2 -20712.394} C_VEL
LIN {X 0,Y 366.291,Z 640.504,A -85,B 0,C 180,E1 -20713.83,E2 -20713.83} C_VEL
LIN {X 0,Y 367.073,Z 628.106,A -85,B 0,C 180,E1 -20715.07,E2 -20715.07} C_VEL
LIN {X 0,Y 367.948,Z 614.644,A -85,B 0,C 180,E1 -20716.166,E2 -20716.166} C_VEL
LIN {X 0,Y 368.574,Z 600.588,A -85,B 0,C 180,E1 -20717.061,E2 -20717.061} C_VEL
LIN {X 0,Y 369.261,Z 585.649,A -85,B 0,C 180,E1 -20717.775,E2 -20717.775} C_VEL
LIN {X 0,Y 369.856,Z 569.337,A -85,B 0,C 180,E1 -20718.316,E2 -20718.316} C_VEL
LIN {X 0,Y 372.769,Z 474.409,A -85,B 0,C 180,E1 -20721.066,E2 -20721.066} C_VEL
LIN {X 0,Y 370.221,Z 444.468,A -85,B 0,C 180,E1 -20722.018,E2 -20722.018} C_VEL
LIN {X 0,Y 370.029,Z 439.502,A -85,B 0,C 180,E1 -20722.194,E2 -20722.194} C_VEL
LIN {X 0,Y 372.104,Z 412.555,A -85,B 0,C 180,E1 -20725.955,E2 -20725.955} C_VEL
LIN {X 0,Y 374.06,Z 388.753,A -85,B 0,C 180,E1 -20729.279,E2 -20729.279} C_VEL
LIN {X 0,Y 369.729,Z 368.642,A -85,B 0,C 180,E1 -20732.382,E2 -20732.382} C_VEL
LIN {X 0,Y 366.065,Z 352.446,A -85,B 0,C 180,E1 -20734.972,E2 -20734.972} C_VEL
LIN {X 0,Y 366.002,Z 352.45,A -85,B 0,C 180,E1 -20738.312,E2 -20738.312} C_VEL
LIN {X 0,Y 365.986,Z 352.45,A -85,B 0,C 180,E1 -20742.056,E2 -20742.056} C_VEL
LIN {X 0,Y 366.031,Z 352.446,A -85,B 0,C 180,E1 -20745.076,E2 -20745.076} C_VEL
LIN {X 0,Y 365.98,Z 352.453,A -85,B 0,C 180,E1 -20748.281,E2 -20748.281} C_VEL
LIN {X 0,Y 366,Z 352.451,A -85,B 0,C 180,E1 -20752.236,E2 -20752.236} C_VEL
LIN {X 0,Y 366.017,Z 352.447,A -85,B 0,C 180,E1 -20755.376,E2 -20755.376} C_VEL
LIN {X 0,Y 365.993,Z 352.445,A -85,B 0,C 180,E1 -20758.887,E2 -20758.887} C_VEL
LIN {X 0,Y 366.025,Z 352.451,A -85,B 0,C 180,E1 -20762.66,E2 -20762.66} C_VEL
LIN {X 0,Y 366.023,Z 352.451,A -85,B 0,C 180,E1 -20766.305,E2 -20766.305} C_VEL
LIN {X 0,Y 366.114,Z 352.441,A -85,B 0,C 180,E1 -20770.146,E2 -20770.146} C_VEL
LIN {X 0,Y 367.06,Z 355.197,A -85,B 0,C 180,E1 -20770.28,E2 -20770.28} C_VEL
LIN {X 0,Y 377.567,Z 379.844,A -85,B 0,C 180,E1 -20771.466,E2 -20771.466} C_VEL
LIN {X 0,Y 378.817,Z 383.167,A -85,B 0,C 180,E1 -20771.61,E2 -20771.61} C_VEL
LIN {X 0,Y 377.438,Z 457.048,A -85,B 0,C 180,E1 -20773.005,E2 -20773.005} C_VEL
LIN {X 0,Y 377.281,Z 474.701,A -85,B 0,C 180,E1 -20773.415,E2 -20773.415} C_VEL
LIN {X 0,Y 376.812,Z 488.75,A -85,B 0,C 180,E1 -20773.948,E2 -20773.948} C_VEL
LIN {X 0,Y 376.084,Z 502.311,A -85,B 0,C 180,E1 -20774.678,E2 -20774.678} C_VEL
LIN {X 0,Y 375.124,Z 514.536,A -85,B 0,C 180,E1 -20775.538,E2 -20775.538} C_VEL
LIN {X 0,Y 374.137,Z 526.523,A -85,B 0,C 180,E1 -20776.604,E2 -20776.604} C_VEL
LIN {X 0,Y 372.969,Z 538.037,A -85,B 0,C 180,E1 -20777.863,E2 -20777.863} C_VEL
LIN {X 0,Y 371.654,Z 547.724,A -85,B 0,C 180,E1 -20779.137,E2 -20779.137} C_VEL
LIN {X 0,Y 370.239,Z 557.863,A -85,B 0,C 180,E1 -20780.746,E2 -20780.746} C_VEL
LIN {X 0,Y 369.019,Z 566.238,A -85,B 0,C 180,E1 -20782.365,E2 -20782.365} C_VEL
LIN {X 0,Y 367.838,Z 574.25,A -85,B 0,C 180,E1 -20784.263,E2 -20784.263} C_VEL
LIN {X 0,Y 366.868,Z 580.716,A -85,B 0,C 180,E1 -20786.169,E2 -20786.169} C_VEL
LIN {X 0,Y 366.117,Z 586.453,A -85,B 0,C 180,E1 -20788.356,E2 -20788.356} C_VEL
LIN {X 0,Y 365.715,Z 589.782,A -85,B 0,C 180,E1 -20790,E2 -20790} C_VEL
LIN {X 0,Y 365.413,Z 592.925,A -85,B 0,C 180,E1 -20792.197,E2 -20792.197} C_VEL
LIN {X 0,Y 365.371,Z 594.788,A -85,B 0,C 180,E1 -20794.522,E2 -20794.522} C_VEL
LIN {X 0,Y 365.5,Z 595.257,A -85,B 0,C 180,E1 -20796.603,E2 -20796.603} C_VEL
LIN {X 0,Y 365.896,Z 594.487,A -85,B 0,C 180,E1 -20798.81,E2 -20798.81} C_VEL
LIN {X 0,Y 366.464,Z 592.412,A -85,B 0,C 180,E1 -20801.019,E2 -20801.019} C_VEL
LIN {X 0,Y 367.567,Z 588.935,A -85,B 0,C 180,E1 -20803.219,E2 -20803.219} C_VEL
LIN {X 0,Y 368.847,Z 583.98,A -85,B 0,C 180,E1 -20805.418,E2 -20805.418} C_VEL
LIN {X 0,Y 370.043,Z 579.152,A -85,B 0,C 180,E1 -20807.062,E2 -20807.062} C_VEL
LIN {X 0,Y 371.663,Z 572.202,A -85,B 0,C 180,E1 -20808.97,E2 -20808.97} C_VEL
LIN {X 0,Y 373.552,Z 563.545,A -85,B 0,C 180,E1 -20810.871,E2 -20810.871} C_VEL
LIN {X 0,Y 375.4,Z 554.451,A -85,B 0,C 180,E1 -20812.489,E2 -20812.489} C_VEL
LIN {X 0,Y 377.249,Z 544.363,A -85,B 0,C 180,E1 -20813.964,E2 -20813.964} C_VEL
LIN {X 0,Y 378.986,Z 533.211,A -85,B 0,C 180,E1 -20815.303,E2 -20815.303} C_VEL
LIN {X 0,Y 380.73,Z 520.817,A -85,B 0,C 180,E1 -20816.496,E2 -20816.496} C_VEL
LIN {X 0,Y 382.029,Z 508.803,A -85,B 0,C 180,E1 -20817.43,E2 -20817.43} C_VEL
LIN {X 0,Y 382.968,Z 496.844,A -85,B 0,C 180,E1 -20818.172,E2 -20818.172} C_VEL
LIN {X 0,Y 383.728,Z 483.262,A -85,B 0,C 180,E1 -20818.801,E2 -20818.801} C_VEL
LIN {X 0,Y 384.094,Z 469.142,A -85,B 0,C 180,E1 -20819.247,E2 -20819.247} C_VEL
LIN {X 0,Y 385.987,Z 392.891,A -85,B 0,C 180,E1 -20820.689,E2 -20820.689} C_VEL
LIN {X 0,Y 377.005,Z 373.826,A -85,B 0,C 180,E1 -20821.843,E2 -20821.843} C_VEL
LIN {X 0,Y 367.32,Z 355.871,A -85,B 0,C 180,E1 -20823.11,E2 -20823.11} C_VEL
LIN {X 0,Y 366.137,Z 353.516,A -85,B 0,C 180,E1 -20823.274,E2 -20823.274} C_VEL
LIN {X 0,Y 365.933,Z 352.461,A -85,B 0,C 180,E1 -20823.323,E2 -20823.323} C_VEL
LIN {X 0,Y 365.947,Z 352.456,A -85,B 0,C 180,E1 -20827.091,E2 -20827.091} C_VEL
LIN {X 0,Y 365.27,Z 352.543,A -85,B 0,C 180,E1 -20828.01,E2 -20828.01} C_VEL
LIN {X 0,Y 362.398,Z 352.901,A -85,B 0,C 180,E1 -20829.504,E2 -20829.504} C_VEL
LIN {X 0,Y 359.981,Z 353.206,A -85,B 0,C 180,E1 -20830.713,E2 -20830.713} C_VEL
LIN {X 0,Y 358.961,Z 353.331,A -85,B 0,C 180,E1 -20831.649,E2 -20831.649} C_VEL
LIN {X 0,Y 358.886,Z 353.338,A -85,B 0,C 180,E1 -20831.966,E2 -20831.966} C_VEL
LIN {X 0,Y 358.934,Z 353.329,A -85,B 0,C 180,E1 -20835.369,E2 -20835.369} C_VEL
LIN {X 0,Y 358.906,Z 353.331,A -85,B 0,C 180,E1 -20838.428,E2 -20838.428} C_VEL
LIN {X 0,Y 358.909,Z 353.315,A -85,B 0,C 180,E1 -20841.353,E2 -20841.353} C_VEL
LIN {X 0,Y 358.917,Z 353.309,A -85,B 0,C 180,E1 -20845.05,E2 -20845.05} C_VEL
LIN {X 0,Y 358.898,Z 353.329,A -85,B 0,C 180,E1 -20848.2,E2 -20848.2} C_VEL
LIN {X 0,Y 358.941,Z 353.329,A -85,B 0,C 180,E1 -20851.42,E2 -20851.42} C_VEL
LIN {X 0,Y 358.964,Z 353.317,A -85,B 0,C 180,E1 -20854.577,E2 -20854.577} C_VEL
LIN {X 0,Y 359.023,Z 353.359,A -85,B 0,C 180,E1 -20857.738,E2 -20857.738} C_VEL
LIN {X 0,Y 365.151,Z 375.964,A -85,B 0,C 180,E1 -20858.574,E2 -20858.574} C_VEL
LIN {X 0,Y 362.72,Z 470.693,A -85,B 0,C 180,E1 -20861.35,E2 -20861.35} C_VEL
LIN {X 0,Y 362.384,Z 486.655,A -85,B 0,C 180,E1 -20862.058,E2 -20862.058} C_VEL
LIN {X 0,Y 361.815,Z 500.763,A -85,B 0,C 180,E1 -20862.901,E2 -20862.901} C_VEL
LIN {X 0,Y 361.2,Z 514.56,A -85,B 0,C 180,E1 -20863.958,E2 -20863.958} C_VEL
LIN {X 0,Y 360.47,Z 527.936,A -85,B 0,C 180,E1 -20865.224,E2 -20865.224} C_VEL
LIN {X 0,Y 359.834,Z 540.152,A -85,B 0,C 180,E1 -20866.634,E2 -20866.634} C_VEL
LIN {X 0,Y 359.211,Z 551.263,A -85,B 0,C 180,E1 -20868.185,E2 -20868.185} C_VEL
LIN {X 0,Y 358.648,Z 561.374,A -85,B 0,C 180,E1 -20869.876,E2 -20869.876} C_VEL
LIN {X 0,Y 358.228,Z 569.809,A -85,B 0,C 180,E1 -20871.567,E2 -20871.567} C_VEL
LIN {X 0,Y 357.941,Z 577.948,A -85,B 0,C 180,E1 -20873.539,E2 -20873.539} C_VEL
LIN {X 0,Y 357.9,Z 584.474,A -85,B 0,C 180,E1 -20875.51,E2 -20875.51} C_VEL
LIN {X 0,Y 357.936,Z 588.63,A -85,B 0,C 180,E1 -20877.052,E2 -20877.052} C_VEL
LIN {X 0,Y 358.102,Z 592.537,A -85,B 0,C 180,E1 -20878.879,E2 -20878.879} C_VEL
LIN {X 0,Y 358.569,Z 595.984,A -85,B 0,C 180,E1 -20881.119,E2 -20881.119} C_VEL
LIN {X 0,Y 359.377,Z 597.936,A -85,B 0,C 180,E1 -20883.352,E2 -20883.352} C_VEL
LIN {X 0,Y 360.544,Z 598.465,A -85,B 0,C 180,E1 -20885.574,E2 -20885.574} C_VEL
LIN {X 0,Y 361.982,Z 597.601,A -85,B 0,C 180,E1 -20887.784,E2 -20887.784} C_VEL
LIN {X 0,Y 363.95,Z 595.292,A -85,B 0,C 180,E1 -20889.974,E2 -20889.974} C_VEL
LIN {X 0,Y 366.531,Z 591.429,A -85,B 0,C 180,E1 -20892.134,E2 -20892.134} C_VEL
LIN {X 0,Y 369.279,Z 585.969,A -85,B 0,C 180,E1 -20894.275,E2 -20894.275} C_VEL
LIN {X 0,Y 371.976,Z 579.885,A -85,B 0,C 180,E1 -20896.091,E2 -20896.091} C_VEL
LIN {X 0,Y 375.049,Z 572.036,A -85,B 0,C 180,E1 -20897.948,E2 -20897.948} C_VEL
LIN {X 0,Y 377.825,Z 563.964,A -85,B 0,C 180,E1 -20899.493,E2 -20899.493} C_VEL
LIN {X 0,Y 380.857,Z 554.245,A -85,B 0,C 180,E1 -20901.016,E2 -20901.016} C_VEL
LIN {X 0,Y 384.104,Z 542.457,A -85,B 0,C 180,E1 -20902.516,E2 -20902.516} C_VEL
LIN {X 0,Y 386.983,Z 530.543,A -85,B 0,C 180,E1 -20903.749,E2 -20903.749} C_VEL
LIN {X 0,Y 389.843,Z 515.855,A -85,B 0,C 180,E1 -20904.975,E2 -20904.975} C_VEL
LIN {X 0,Y 391.885,Z 502.916,A -85,B 0,C 180,E1 -20905.834,E2 -20905.834} C_VEL
LIN {X 0,Y 393.565,Z 488.689,A -85,B 0,C 180,E1 -20906.575,E2 -20906.575} C_VEL
LIN {X 0,Y 395.745,Z 465.85,A -85,B 0,C 180,E1 -20907.435,E2 -20907.435} C_VEL
LIN {X 0,Y 402.054,Z 413.665,A -85,B 0,C 180,E1 -20909.13,E2 -20909.13} C_VEL
LIN {X 0,Y 398.052,Z 405.751,A -85,B 0,C 180,E1 -20910.569,E2 -20910.569} C_VEL
LIN {X 0,Y 394.273,Z 399.117,A -85,B 0,C 180,E1 -20912.076,E2 -20912.076} C_VEL
LIN {X 0,Y 391.684,Z 394.968,A -85,B 0,C 180,E1 -20913.233,E2 -20913.233} C_VEL
LIN {X 0,Y 389.548,Z 391.577,A -85,B 0,C 180,E1 -20914.287,E2 -20914.287} C_VEL
LIN {X 0,Y 387.288,Z 388.141,A -85,B 0,C 180,E1 -20915.579,E2 -20915.579} C_VEL
LIN {X 0,Y 386.441,Z 386.997,A -85,B 0,C 180,E1 -20916.113,E2 -20916.113} C_VEL
LIN {X 0,Y 384.261,Z 383.968,A -85,B 0,C 180,E1 -20917.738,E2 -20917.738} C_VEL
LIN {X 0,Y 383.511,Z 382.522,A -85,B 0,C 180,E1 -20918.491,E2 -20918.491} C_VEL
LIN {X 0,Y 381.206,Z 380.697,A -85,B 0,C 180,E1 -20921.413,E2 -20921.413} C_VEL
LIN {X 0,Y 380.777,Z 380.214,A -85,B 0,C 180,E1 -20922.892,E2 -20922.892} C_VEL
LIN {X 0,Y 381.077,Z 380.617,A -85,B 0,C 180,E1 -20925.286,E2 -20925.286} C_VEL
LIN {X 0,Y 383.071,Z 382.405,A -85,B 0,C 180,E1 -20928.075,E2 -20928.075} C_VEL
LIN {X 0,Y 383.471,Z 382.917,A -85,B 0,C 180,E1 -20928.495,E2 -20928.495} C_VEL
LIN {X 0,Y 384.983,Z 385.856,A -85,B 0,C 180,E1 -20929.933,E2 -20929.933} C_VEL
LIN {X 0,Y 386.783,Z 387.857,A -85,B 0,C 180,E1 -20931.142,E2 -20931.142} C_VEL
LIN {X 0,Y 387.596,Z 389.969,A -85,B 0,C 180,E1 -20931.739,E2 -20931.739} C_VEL
LIN {X 0,Y 389.518,Z 398.512,A -85,B 0,C 180,E1 -20933.361,E2 -20933.361} C_VEL
LIN {X 0,Y 392.679,Z 412.836,A -85,B 0,C 180,E1 -20935.531,E2 -20935.531} C_VEL
LIN {X 0,Y 393.149,Z 415.968,A -85,B 0,C 180,E1 -20935.884,E2 -20935.884} C_VEL
LIN {X 0,Y 393.995,Z 436.558,A -85,B 0,C 180,E1 -20937.506,E2 -20937.506} C_VEL
LIN {X 0,Y 394.631,Z 457.182,A -85,B 0,C 180,E1 -20938.926,E2 -20938.926} C_VEL
LIN {X 0,Y 394.754,Z 473.678,A -85,B 0,C 180,E1 -20939.889,E2 -20939.889} C_VEL
LIN {X 0,Y 394.214,Z 488.202,A -85,B 0,C 180,E1 -20940.579,E2 -20940.579} C_VEL
LIN {X 0,Y 388.287,Z 540.512,A -85,B 0,C 180,E1 -20942.285,E2 -20942.285} C_VEL
LIN {X 0,Y 385.556,Z 556.975,A -85,B 0,C 180,E1 -20942.988,E2 -20942.988} C_VEL
LIN {X 0,Y 382.65,Z 571.184,A -85,B 0,C 180,E1 -20943.793,E2 -20943.793} C_VEL
LIN {X 0,Y 379.022,Z 585.879,A -85,B 0,C 180,E1 -20944.846,E2 -20944.846} C_VEL
LIN {X 0,Y 375.392,Z 599.255,A -85,B 0,C 180,E1 -20946.056,E2 -20946.056} C_VEL
LIN {X 0,Y 371.939,Z 611.167,A -85,B 0,C 180,E1 -20947.392,E2 -20947.392} C_VEL
LIN {X 0,Y 368.72,Z 621.757,A -85,B 0,C 180,E1 -20948.842,E2 -20948.842} C_VEL
LIN {X 0,Y 365.376,Z 632.78,A -85,B 0,C 180,E1 -20950.689,E2 -20950.689} C_VEL
LIN {X 0,Y 362.507,Z 641.932,A -85,B 0,C 180,E1 -20952.572,E2 -20952.572} C_VEL
LIN {X 0,Y 360.138,Z 650.375,A -85,B 0,C 180,E1 -20954.777,E2 -20954.777} C_VEL
LIN {X 0,Y 358.558,Z 657.111,A -85,B 0,C 180,E1 -20957.017,E2 -20957.017} C_VEL
LIN {X 0,Y 357.731,Z 661.682,A -85,B 0,C 180,E1 -20958.923,E2 -20958.923} C_VEL
LIN {X 0,Y 357.28,Z 672.047,A -85,B 0,C 180,E1 -20960.692,E2 -20960.692} C_VEL
LIN {X 0,Y 356.874,Z 680.211,A -85,B 0,C 180,E1 -20962.387,E2 -20962.387} C_VEL
